				JMP START;			
			END_IF
		ELSE
			IF _Command.ExecuteDataReturn(ADR(_ExecutionParameters.CommandText), SIZEOF(_ExecutionParameters.CommandText), ADR(_SQLResult)) THEN
				IF _Command.bError THEN
					_GetError := TRUE;
					_Logger := _Command.ipTcResult;
					_State := DB_COMMAND_EXECUTION_STATE.DISCONNECTING;
				ELSE
					_State := DB_COMMAND_EXECUTION_STATE.LOADING_RESULT_DATA_SET;
				END_IF
				
				JMP START;			
			END_IF
		END_IF
		
	DB_COMMAND_EXECUTION_STATE.LOADING_RESULT_DATA_SET:
		IF _SQLResult.Read(0, _ExecutionParameters.MaxRecordsToReadAtTime, _ExecutionParameters.TargetBuffer, _ExecutionParameters.TargetBufferSize, TRUE, TRUE) THEN			
			IF _SQLResult.bError THEN
				_GetError := TRUE;
				_SQLResult.Release();
				_Logger := _SQLResult.ipTcResult;
			ELSE
				_DataSetLoaded := TRUE;
			END_IF

			_State := DB_COMMAND_EXECUTION_STATE.DISCONNECTING;
			
			JMP START;			
		END_IF

	DB_COMMAND_EXECUTION_STATE.DISCONNECTING:
		CASE _DisconnectingState OF
			DB_COMMAND_DISCONNECTING_STATE.IDLING:
				IF _DataSetLoaded THEN
					_DisconnectingState := DB_COMMAND_DISCONNECTING_STATE.DATA_SET_RELEASING;
				ELSIF _Connected THEN
					_DisconnectingState := DB_COMMAND_DISCONNECTING_STATE.DISCONNECTING;					
				ELSE
					_State := DB_COMMAND_EXECUTION_STATE.IDLING;	
					_Done := _LastException.Empty;	
				END_IF
				
				JMP START;
				
			DB_COMMAND_DISCONNECTING_STATE.DATA_SET_RELEASING:
				IF _SQLResult.Release() THEN
					_DataSetLoaded := FALSE;
					_DisconnectingState := DB_COMMAND_DISCONNECTING_STATE.DISCONNECTING;
					JMP START;										
				END_IF
				
			DB_COMMAND_DISCONNECTING_STATE.DISCONNECTING:
				IF _DbConnection.Disconnect() THEN
					_Connected := FALSE;
					_DisconnectingState := DB_COMMAND_DISCONNECTING_STATE.IDLING;
					JMP START;										
				END_IF
		END_CASE	
END_CASE
END_METHOD

{attribute 'monitoring' := 'call'}
{attribute 'OPC.UA.DA.Property' := '1'}
{attribute 'OPC.UA.DA.Access' := '1'}
PROPERTY LastException : REFERENCE TO Exception
GET
LastException REF= _LastException;
END_GET
END_PROPERTY

METHOD Reset
VAR_OUTPUT
	exception : Exception;
END_VAR
IF Busy THEN
	_LastExceptionHelper.Throw(0, "Previous command execution is not finished", __POUNAME(), ClassName, CurrentNamespace.Name, __POSITION()); 
	RETURN;
END_IF

_Done := FALSE;
_State := DB_COMMAND_EXECUTION_STATE.STARTING;
_GetError := FALSE;
_Logger := 0;	
_Connected := FALSE;
_DataSetLoaded := FALSE;
_DisconnectingState := DB_COMMAND_DISCONNECTING_STATE.IDLING;
_LastException.Clear();
END_METHOD

METHOD Start 
VAR_INPUT
	dbId : UDINT;
	commandText : Tc2_System.T_MaxString;
	targetBuffer : PVOID;
	targetBufferSize : UDINT;
	maxRecordsToReadAtTime : UINT;
END_VAR
VAR_OUTPUT
	exception : Exception;
END_VAR
VAR
	executionParameters : POINTER TO DB_COMMAND_EXECUTION_PARAMETERS;
END_VAR
IF Busy THEN
	_LastExceptionHelper.Throw(0, "Previous command execution is not finished", __POUNAME(), ClassName, CurrentNamespace.Name, __POSITION()); 
	RETURN;
END_IF

IF maxRecordsToReadAtTime > 0 AND_THEN (targetBuffer = 0 OR_ELSE targetBufferSize = 0) THEN
	_LastExceptionHelper.Throw(0, "Parameter 'maxRecordsToReadAtTime' is greater then zero, but 'targetBuffer' or 'targetBufferSize' has incorrect values", __POUNAME(), ClassName, CurrentNamespace.Name, __POSITION()); 
	RETURN;
END_IF

_ExecutionParameters.DbId := dbId;
_ExecutionParameters.CommandText := commandText;
_ExecutionParameters.TargetBuffer := targetBuffer; 
_ExecutionParameters.TargetBufferSize := targetBufferSize;
_ExecutionParameters.MaxRecordsToReadAtTime := maxRecordsToReadAtTime;

Reset();
END_METHOD

{attribute 'monitoring' := 'call'}
{attribute 'OPC.UA.DA.Property' := '1'}
{attribute 'OPC.UA.DA.Access' := '1'}
PROPERTY State : DB_COMMAND_EXECUTION_STATE
GET
State := _State;
END_GET
END_PROPERTY

{attribute 'monitoring' := 'call'}
{attribute 'OPC.UA.DA.Property' := '1'}
{attribute 'OPC.UA.DA.Access' := '1'}
PROPERTY Timeout : TIME
GET
Timeout := _Command.tTimeout;
END_GET
SET
_Command.tTimeout := Timeout;
_SQLResult.tTimeout := Timeout;
END_SET
END_PROPERTY

END_FUNCTION_BLOCK

// ---- Database/StoredProcedure/DbProcedureExecutor.TcPOU
{attribute 'no_explicit_call' := 'do not call this function block directly'} 
FUNCTION_BLOCK DbProcedureExecutor EXTENDS TC.ToolkitObject IMPLEMENTS TC.IAction
VAR	
	_ClassName : STRING := __POUNAME();

	_DbConnection : Tc3_Database.FB_SQLDatabaseEvt(sNetID := '', tTimeout := T#10S);	

	_ExecutionParameters : DB_ROCEDURE_EXECUTION_PARAMETERS;

	_StoredProcedure : Tc3_Database.FB_SQLStoredProcedureEvt(sNetID:='', tTimeout := T#10S);
	_SQLResult: Tc3_Database.FB_SQLResultEvt(sNetID := '', tTimeout := T#10S);
	
	_Done : BOOL;
	_State : DB_PROCEDURE_EXECUTION_STATE;
	_GetError : BOOL;
	_Logger : Tc3_EventLogger.I_TcMessage;	
	_Connected : BOOL;
	_Prepared : BOOL;
	_DataSetLoaded : BOOL;
	_DisconnectingState : DB_PROCEDURE_DISCONNECTING_STATE;
	_LastException : Exception;
END_VAR

{attribute 'monitoring' := 'call'}
{attribute 'OPC.UA.DA.Property' := '1'}
{attribute 'OPC.UA.DA.Access' := '1'}
PROPERTY Busy : BOOL
GET
Busy := State <> DB_PROCEDURE_EXECUTION_STATE.IDLING;
END_GET
END_PROPERTY

{attribute 'monitoring' := 'call'}
PROPERTY ClassName : STRING
GET
ClassName := _ClassName;
END_GET
END_PROPERTY

{attribute 'monitoring' := 'call'}
{attribute 'OPC.UA.DA.Property' := '1'}
{attribute 'OPC.UA.DA.Access' := '1'}
PROPERTY Done : BOOL
GET
Done := _Done;
END_GET
END_PROPERTY

{attribute 'monitoring' := 'call'}
{attribute 'OPC.UA.DA.Property' := '1'}
{attribute 'OPC.UA.DA.Access' := '1'}
PROPERTY Error : BOOL
GET
Error := State = DB_PROCEDURE_EXECUTION_STATE.IDLING AND_THEN NOT _LastException.Empty;
END_GET
END_PROPERTY

METHOD Execute
VAR
	requestEventTextError : BOOL;
	requestEventTextErrorCode : HRESULT;
END_VAR
VAR_INST
	errorMessage : STRING(255);	
END_VAR
START:

IF NOT _LastException.Empty THEN
	_GetError := FALSE;
END_IF

IF _GetError THEN
	IF _Logger <> 0 THEN 
		IF _Logger.RequestEventText(1033, errorMessage, SIZEOF(errorMessage), bError => requestEventTextError, hrErrorCode => requestEventTextErrorCode) THEN
			IF requestEventTextError THEN					
				errorMessage := StringHelper.Concat2('_Logger.RequestEventText() call error. Error code is ', TO_STRING(requestEventTextErrorCode));
			END_IF
		ELSE
			RETURN;
		END_IF			
	ELSE
		errorMessage :=  'Logger is not specified';
	END_IF				
	
	_LastExceptionHelper.Throw(0, TO_WSTRING(errorMessage), __POUNAME(), ClassName, CurrentNamespace.Name, __POSITION());
	JMP START;	
END_IF

CASE State OF
	DB_PROCEDURE_EXECUTION_STATE.STARTING:
		MEMSET(_ExecutionParameters.TargetBuffer, 0, _ExecutionParameters.TargetBufferSize);	
		_State := DB_PROCEDURE_EXECUTION_STATE.CONNECTING;			
		JMP START;
				
	DB_PROCEDURE_EXECUTION_STATE.CONNECTING:
		IF _DbConnection.Connect(hDBID := _ExecutionParameters.DBID) THEN
			IF _DbConnection.bError THEN
				_GetError := TRUE;
				_Logger := _DbConnection.ipTcResult;
				_State := DB_PROCEDURE_EXECUTION_STATE.DISCONNECTING;				
			ELSE
				_Connected := TRUE;
				_State := DB_PROCEDURE_EXECUTION_STATE.PREPARING;
			END_IF			

			JMP START;
		END_IF
	
	DB_PROCEDURE_EXECUTION_STATE.PREPARING:
		IF _DbConnection.CreateSP(sProcedureName := _ExecutionParameters.ProcedureName, pParameterInfo := _ExecutionParameters.ParameterDescriptors, cbParameterInfo := _ExecutionParameters.ParameterDescriptorsSize, pSQLProcedure := ADR(_StoredProcedure)) THEN
			IF _DbConnection.bError THEN
				_GetError := TRUE;
				_Logger := _DbConnection.ipTcResult;
				_State := DB_PROCEDURE_EXECUTION_STATE.DISCONNECTING;				
			ELSE
				_Prepared := TRUE;
				_State := DB_PROCEDURE_EXECUTION_STATE.EXECUTING;
			END_IF
			
			JMP START;
		END_IF
	
	DB_PROCEDURE_EXECUTION_STATE.EXECUTING:
		IF _ExecutionParameters.MaxRecordsToReadAtTime = 0 THEN
			IF _StoredProcedure.Execute(_ExecutionParameters.ParameterValues, _ExecutionParameters.ParameterValuesSize) THEN
				IF _StoredProcedure.bError THEN
					_GetError := TRUE;
					_Logger := _StoredProcedure.ipTcResult;
				END_IF
				
				_State := DB_PROCEDURE_EXECUTION_STATE.DISCONNECTING;
				
				JMP START;			
			END_IF
		ELSE
			IF _StoredProcedure.ExecuteDataReturn(_ExecutionParameters.ParameterValues, _ExecutionParameters.ParameterValuesSize, ADR(_SQLResult)) THEN
				IF _StoredProcedure.bError THEN
					_GetError := TRUE;
					_Logger := _StoredProcedure.ipTcResult;
					_State := DB_PROCEDURE_EXECUTION_STATE.DISCONNECTING;
				ELSE
					_State := DB_PROCEDURE_EXECUTION_STATE.LOADING_RESULT_DATA_SET;
				END_IF
								
				JMP START;			
			END_IF
		END_IF
		
	DB_PROCEDURE_EXECUTION_STATE.LOADING_RESULT_DATA_SET:
		IF _SQLResult.Read(0, _ExecutionParameters.MaxRecordsToReadAtTime, _ExecutionParameters.TargetBuffer, _ExecutionParameters.TargetBufferSize, TRUE, TRUE) THEN
			IF _SQLResult.bError THEN
				_GetError := TRUE;
				_SQLResult.Release();
				_Logger := _SQLResult.ipTcResult;
			ELSE				
				_DataSetLoaded := TRUE;
			END_IF
			
			_State := DB_PROCEDURE_EXECUTION_STATE.DISCONNECTING;
			
			JMP START;			
		END_IF		

	DB_PROCEDURE_EXECUTION_STATE.DISCONNECTING:
		CASE _DisconnectingState OF
			DB_PROCEDURE_DISCONNECTING_STATE.IDLING:				
				IF _DataSetLoaded THEN
					_DisconnectingState := DB_PROCEDURE_DISCONNECTING_STATE.DATA_SET_RELEASING;
				ELSIF _Prepared THEN
					_DisconnectingState := DB_PROCEDURE_DISCONNECTING_STATE.PARAMETERS_RELEASING;					
				ELSIF _Connected THEN
					_DisconnectingState := DB_PROCEDURE_DISCONNECTING_STATE.DISCONNECTING;					
				ELSE
					_State := DB_PROCEDURE_EXECUTION_STATE.IDLING;				
					_Done := _LastException.Empty;	
				END_IF
				
				JMP START;
				
			DB_PROCEDURE_DISCONNECTING_STATE.DATA_SET_RELEASING:
				IF _SQLResult.Release() THEN
					_DataSetLoaded := FALSE;
					_DisconnectingState := DB_PROCEDURE_DISCONNECTING_STATE.PARAMETERS_RELEASING;
					JMP START;					
				END_IF
			
			DB_PROCEDURE_DISCONNECTING_STATE.PARAMETERS_RELEASING:
				IF _StoredProcedure.Release() THEN
					_Prepared := FALSE;
					_DisconnectingState := DB_PROCEDURE_DISCONNECTING_STATE.DISCONNECTING;
					JMP START;										
				END_IF
				
			DB_PROCEDURE_DISCONNECTING_STATE.DISCONNECTING:
				IF _DbConnection.Disconnect() THEN
					_Connected := FALSE;
					_DisconnectingState := DB_PROCEDURE_DISCONNECTING_STATE.IDLING;
					JMP START;										
				END_IF
		END_CASE	
END_CASE
END_METHOD

{attribute 'monitoring' := 'call'}
{attribute 'OPC.UA.DA.Property' := '1'}
{attribute 'OPC.UA.DA.Access' := '1'}
PROPERTY LastException : REFERENCE TO Exception
GET
LastException REF= _LastException;
END_GET
END_PROPERTY

{attribute 'OPC.UA.DA.Property' := '1'}
{attribute 'OPC.UA.DA.Access' := '1'}
{attribute 'monitoring' := 'call'}
PROPERTY ProcedureName : REFERENCE TO Tc2_System.T_MaxString
GET
ProcedureName REF= _ExecutionParameters.ProcedureName;
END_GET
END_PROPERTY

METHOD Reset 
VAR_OUTPUT
	exception : Exception;
END_VAR
IF Busy THEN
	_LastExceptionHelper.Throw(0, "Previous command execution is not finished", __POUNAME(), ClassName, CurrentNamespace.Name, __POSITION()); 
	RETURN;
END_IF

_Done := FALSE;
_State := DB_PROCEDURE_EXECUTION_STATE.STARTING;
_GetError := FALSE;
_Logger := 0;	
_Connected := FALSE;
_Prepared := FALSE;
_DataSetLoaded := FALSE;
_DisconnectingState := DB_PROCEDURE_DISCONNECTING_STATE.IDLING;
_LastException.Clear();
END_METHOD

METHOD Start 
VAR_INPUT
	dbId : UDINT;
	procedureName : Tc2_System.T_MaxString;
	parameterDescriptors : POINTER TO Tc3_Database.ST_SQLSPParameter;
	parameterDescriptorsSize : UDINT;
	parameterValues : PVOID;
	parameterValuesSize : UDINT;
	targetBuffer : PVOID;
	targetBufferSize : UDINT;
	maxRecordsToReadAtTime : UINT;
END_VAR
VAR_OUTPUT
	exception : Exception;
END_VAR
IF Busy THEN
	_LastExceptionHelper.Throw(0, "Previous command execution is not finished", __POUNAME(), ClassName, CurrentNamespace.Name, __POSITION()); 
	RETURN;
END_IF

IF maxRecordsToReadAtTime > 0 AND_THEN (targetBuffer = 0 OR_ELSE targetBufferSize = 0) THEN
	_LastExceptionHelper.Throw(0, "Parameter 'maxRecordsToReadAtTime' is greater then zero, but 'targetBuffer' or 'targetBufferSize' has incorrect values", __POUNAME(), ClassName, CurrentNamespace.Name, __POSITION()); 
	RETURN;
END_IF

_ExecutionParameters.DbId := dbId;
_ExecutionParameters.ProcedureName := procedureName;
_ExecutionParameters.ParameterDescriptors := parameterDescriptors;
_ExecutionParameters.ParameterDescriptorsSize := parameterDescriptorsSize;
_ExecutionParameters.ParameterValues := parameterValues;
_ExecutionParameters.ParameterValuesSize := parameterValuesSize;
_ExecutionParameters.TargetBuffer := targetBuffer; 
_ExecutionParameters.TargetBufferSize := targetBufferSize;
_ExecutionParameters.MaxRecordsToReadAtTime := maxRecordsToReadAtTime;

Reset();
END_METHOD

{attribute 'monitoring' := 'call'}
{attribute 'OPC.UA.DA.Property' := '1'}
{attribute 'OPC.UA.DA.Access' := '1'}
PROPERTY State : DB_PROCEDURE_EXECUTION_STATE
GET
State := _State;
END_GET
END_PROPERTY

{attribute 'monitoring' := 'call'}
{attribute 'OPC.UA.DA.Property' := '1'}
{attribute 'OPC.UA.DA.Access' := '1'}
PROPERTY Timeout : TIME
GET
Timeout := _StoredProcedure.tTimeout;
END_GET
SET
_StoredProcedure.tTimeout := Timeout;
_SQLResult.tTimeout := Timeout;
END_SET
END_PROPERTY

END_FUNCTION_BLOCK

// ---- Files/CreateDirectory.TcPOU
{attribute 'no_explicit_call' := 'do not call this function block directly'} 
FUNCTION_BLOCK CreateDirectory EXTENDS ToolkitObject IMPLEMENTS IAction
VAR
	{attribute 'OPC.UA.DA' := '0'}
	_ClassName : STRING := __POUNAME();

	{attribute 'OPC.UA.DA' := '0'}
    _CreateDirectory : Tc2_System.FB_CreateDir;
	
	{attribute 'OPC.UA.DA' := '0'}
	_NeedStart : BOOL;
	{attribute 'OPC.UA.DA' := '0'}
	_Done : BOOL;
END_VAR

{attribute 'monitoring' := 'call'}
{attribute 'OPC.UA.DA.Property' := '1'}
{attribute 'OPC.UA.DA' := '1'}
PROPERTY AmsNetId : Tc2_System.T_AmsNetID
GET
AmsNetId := _CreateDirectory.sNetId;
END_GET
SET
_CreateDirectory.sNetId := AmsNetId;
END_SET
END_PROPERTY

{attribute 'monitoring' := 'call'}
{attribute 'OPC.UA.DA.Property' := '1'}
{attribute 'OPC.UA.DA.Access' := '1'}
PROPERTY Busy : BOOL
GET
Busy := _NeedStart OR_ELSE _CreateDirectory.bBusy;
END_GET
END_PROPERTY

{attribute 'monitoring' := 'call'}
PROPERTY ClassName : STRING
GET
ClassName := _ClassName;
END_GET
END_PROPERTY

{attribute 'monitoring' := 'call'}
{attribute 'OPC.UA.DA.Property' := '1'}
{attribute 'OPC.UA.DA.Access' := '1'}
PROPERTY Done : BOOL
GET
Done := _Done;
END_GET
END_PROPERTY

{attribute 'monitoring' := 'call'}
{attribute 'OPC.UA.DA.Property' := '1'}
{attribute 'OPC.UA.DA.Access' := '1'}
PROPERTY Error : BOOL
GET
Error := _CreateDirectory.bError;
END_GET
END_PROPERTY

METHOD Execute
VAR
	message : ERROR_MESSAGE;
END_VAR
IF _NeedStart OR_ELSE _CreateDirectory.bBusy THEN
	_CreateDirectory(bExecute := TRUE);
	_NeedStart := FALSE;
	
	IF _CreateDirectory.bError THEN
		message := "An error occurred while creating the directory '";
		WStringHelper.Append2(message, TO_WSTRING(_CreateDirectory.sPathName), "'");	
		_LastException.Configure(message, __POUNAME(), ClassName, CurrentNamespace.Name, __POSITION(), _CreateDirectory.nErrId).Throw();
	ELSIF NOT _CreateDirectory.bBusy THEN
		_Done := TRUE;
	END_IF
END_IF
END_METHOD

{attribute 'monitoring' := 'call'}
{attribute 'OPC.UA.DA.Property' := '1'}
{attribute 'OPC.UA.DA.Access' := '1'}
PROPERTY LastException : REFERENCE TO Exception
GET
LastException REF= _LastException;
END_GET
END_PROPERTY

{attribute 'monitoring' := 'call'}
{attribute 'OPC.UA.DA.Property' := '1'}
{attribute 'OPC.UA.DA' := '1'}
PROPERTY PathType : Tc2_System.E_OpenPath
GET
PathType := _CreateDirectory.ePath;
END_GET
SET
_CreateDirectory.ePath := PathType;
END_SET
END_PROPERTY

METHOD Start
VAR_INPUT
	directoryPath : Tc2_System.T_MaxString;
END_VAR
_NeedStart := TRUE;
_Done := FALSE;
_CreateDirectory.sPathName := directoryPath;

_LastException.Clear();
END_METHOD

{attribute 'monitoring' := 'call'}
{attribute 'OPC.UA.DA.Property' := '1'}
{attribute 'OPC.UA.DA' := '1'}
PROPERTY Timeout : TIME
GET
Timeout := _CreateDirectory.tTimeout;
END_GET
SET
_CreateDirectory.tTimeout := Timeout;
END_SET
END_PROPERTY

END_FUNCTION_BLOCK

// ---- Files/DeleteDirectory.TcPOU
{attribute 'no_explicit_call' := 'do not call this function block directly'} 
FUNCTION_BLOCK DeleteDirectory EXTENDS ToolkitObject IMPLEMENTS IAction
VAR
	{attribute 'OPC.UA.DA' := '0'}
	_ClassName : STRING := __POUNAME();

	{attribute 'OPC.UA.DA' := '0'}
    _DeleteDirectory : Tc2_System.FB_RemoveDir;	
	
	{attribute 'OPC.UA.DA' := '0'}
	_NeedStart : BOOL;
	{attribute 'OPC.UA.DA' := '0'}
	_Done : BOOL;
END_VAR

{attribute 'monitoring' := 'call'}
{attribute 'OPC.UA.DA.Property' := '1'}
{attribute 'OPC.UA.DA' := '1'}
PROPERTY AmsNetId : Tc2_System.T_AmsNetID
GET
AmsNetId := _DeleteDirectory.sNetId;
END_GET
SET
_DeleteDirectory.sNetId := AmsNetId;
END_SET
END_PROPERTY

{attribute 'monitoring' := 'call'}
{attribute 'OPC.UA.DA.Property' := '1'}
{attribute 'OPC.UA.DA.Access' := '1'}
PROPERTY Busy : BOOL
GET
Busy := _NeedStart OR_ELSE _DeleteDirectory.bBusy;
END_GET
END_PROPERTY

{attribute 'monitoring' := 'call'}
PROPERTY ClassName : STRING
GET
ClassName := _ClassName;
END_GET
END_PROPERTY

{attribute 'monitoring' := 'call'}
{attribute 'OPC.UA.DA.Property' := '1'}
{attribute 'OPC.UA.DA.Access' := '1'}
PROPERTY Done : BOOL
GET
Done := _Done;
END_GET
END_PROPERTY

{attribute 'monitoring' := 'call'}
{attribute 'OPC.UA.DA.Property' := '1'}
{attribute 'OPC.UA.DA.Access' := '1'}
PROPERTY Error : BOOL
GET
Error := _DeleteDirectory.bError;
END_GET
END_PROPERTY

METHOD Execute
VAR
	errorMessage : ERROR_MESSAGE;
END_VAR
IF _NeedStart OR_ELSE _DeleteDirectory.bBusy THEN
	_DeleteDirectory(bExecute := TRUE);
	_NeedStart := FALSE;
	
	IF _DeleteDirectory.bError THEN
		errorMessage := "An error occurred while deleting the directory '";
		WStringHelper.Append2(errorMessage, TO_WSTRING(_DeleteDirectory.sPathName), "'");	
		_LastException.Configure(errorMessage, __POUNAME(), ClassName, CurrentNamespace.Name, __POSITION(), _DeleteDirectory.nErrId).Throw();
	ELSIF NOT _DeleteDirectory.bBusy THEN
		_Done := TRUE;
	END_IF
END_IF
END_METHOD

{attribute 'monitoring' := 'call'}
{attribute 'OPC.UA.DA.Property' := '1'}
{attribute 'OPC.UA.DA.Access' := '1'}
PROPERTY LastException : REFERENCE TO Exception
GET
LastException REF= _LastException;
END_GET
END_PROPERTY

{attribute 'monitoring' := 'call'}
{attribute 'OPC.UA.DA.Property' := '1'}
{attribute 'OPC.UA.DA' := '1'}
PROPERTY PathType : Tc2_System.E_OpenPath
GET
PathType := _DeleteDirectory.ePath;
END_GET
SET
_DeleteDirectory.ePath := PathType;
END_SET
END_PROPERTY

METHOD Start
VAR_INPUT
	directoryPath : Tc2_System.T_MaxString;
END_VAR
_NeedStart := TRUE;
_Done := FALSE;
_DeleteDirectory.sPathName := directoryPath;

_LastException.Clear();
END_METHOD

{attribute 'monitoring' := 'call'}
{attribute 'OPC.UA.DA.Property' := '1'}
{attribute 'OPC.UA.DA' := '1'}
PROPERTY Timeout : TIME
GET
Timeout := _DeleteDirectory.tTimeout;
END_GET
SET
_DeleteDirectory.tTimeout := Timeout;
END_SET
END_PROPERTY

END_FUNCTION_BLOCK

// ---- Files/DeleteFile.TcPOU
{attribute 'no_explicit_call' := 'do not call this function block directly'} 
FUNCTION_BLOCK DeleteFile EXTENDS ToolkitObject IMPLEMENTS IAction
VAR
	{attribute 'OPC.UA.DA' := '0'}
	_ClassName : STRING := __POUNAME();

	{attribute 'OPC.UA.DA' := '0'}
    _Delete : Tc2_System.FB_FileDelete;
	
	{attribute 'OPC.UA.DA' := '0'}
	_NeedStart : BOOL;
	{attribute 'OPC.UA.DA' := '0'}
	_Done : BOOL;
END_VAR

{attribute 'monitoring' := 'call'}
{attribute 'OPC.UA.DA.Property' := '1'}
{attribute 'OPC.UA.DA' := '1'}
PROPERTY AmsNetId : Tc2_System.T_AmsNetID
GET
AmsNetId := _Delete.sNetId;
END_GET
SET
_Delete.sNetId := AmsNetId;
END_SET
END_PROPERTY

{attribute 'monitoring' := 'call'}
{attribute 'OPC.UA.DA.Property' := '1'}
{attribute 'OPC.UA.DA.Access' := '1'}
PROPERTY Busy : BOOL
GET
Busy := _NeedStart OR_ELSE _Delete.bBusy;
END_GET
END_PROPERTY

{attribute 'monitoring' := 'call'}
PROPERTY ClassName : STRING
GET
ClassName := _ClassName;
END_GET
END_PROPERTY

{attribute 'monitoring' := 'call'}
{attribute 'OPC.UA.DA.Property' := '1'}
{attribute 'OPC.UA.DA.Access' := '1'}
PROPERTY Done : BOOL
GET
Done := _Done;
END_GET
END_PROPERTY

{attribute 'monitoring' := 'call'}
{attribute 'OPC.UA.DA.Property' := '1'}
{attribute 'OPC.UA.DA.Access' := '1'}
PROPERTY Error : BOOL
GET
Error := _Delete.bError;
END_GET
END_PROPERTY

METHOD Execute
VAR
	message : ERROR_MESSAGE;
END_VAR
IF _NeedStart OR_ELSE _Delete.bBusy THEN
	_Delete(bExecute := TRUE);
	_NeedStart := FALSE;
	
	IF _Delete.bError THEN
		message := "An error occurred while creating the file '";
		WStringHelper.Append2(message, TO_WSTRING(_Delete.sPathName), "'");	
		_LastException.Configure(message, __POUNAME(), ClassName, CurrentNamespace.Name, __POSITION(), _Delete.nErrId).Throw();
	ELSIF NOT _Delete.bBusy THEN
		_Done := TRUE;
	END_IF
END_IF
END_METHOD

{attribute 'monitoring' := 'call'}
{attribute 'OPC.UA.DA.Property' := '1'}
{attribute 'OPC.UA.DA.Access' := '1'}
PROPERTY LastException : REFERENCE TO Exception
GET
LastException REF= _LastException;
END_GET
END_PROPERTY

{attribute 'monitoring' := 'call'}
{attribute 'OPC.UA.DA.Property' := '1'}
{attribute 'OPC.UA.DA' := '1'}
PROPERTY PathType : Tc2_System.E_OpenPath
GET
PathType := _Delete.ePath;
END_GET
SET
_Delete.ePath := PathType;
END_SET
END_PROPERTY

METHOD Start
VAR_INPUT
	filePath : Tc2_System.T_MaxString;
END_VAR
_NeedStart := TRUE;
_Done := FALSE;
_Delete.sPathName := filePath;

_LastException.Clear();
END_METHOD

{attribute 'monitoring' := 'call'}
{attribute 'OPC.UA.DA.Property' := '1'}
{attribute 'OPC.UA.DA' := '1'}
PROPERTY Timeout : TIME
GET
Timeout := _Delete.tTimeout;
END_GET
SET
_Delete.tTimeout := Timeout;
END_SET
END_PROPERTY

END_FUNCTION_BLOCK

// ---- Files/FileContentManager/FileContentManager.TcPOU
{attribute 'no_explicit_call' := 'do not call this function block directly'} 
FUNCTION_BLOCK FileContentManager EXTENDS ToolkitObject IMPLEMENTS IAbortableProcess
VAR
	_ClassName : STRING := __POUNAME();

	_FilePath : Tc2_System.T_MaxString;	
	_OpenMode : FILE_OPEN_MODE;
	_ContentHandlingMode : FILE_CONTENT_HANDLING_MODE;
	_PathType : E_OpenPath;	
	_AmsNetId : Tc2_System.T_AmsNetID;
	_FileHandle : UINT;
		
	_TaskExecutor : SequentialTaskExecutor;
END_VAR

{attribute 'monitoring' := 'call'}
{attribute 'OPC.UA.DA.Property' := '1'}
{attribute 'OPC.UA.DA.Access' := '1'}
PROPERTY FINAL Aborted : BOOL
GET
Aborted := _TaskExecutor.Aborted;
END_GET
END_PROPERTY

{attribute 'monitoring' := 'call'}
{attribute 'OPC.UA.DA.Property' := '1'}
{attribute 'OPC.UA.DA.Access' := '1'}
PROPERTY FINAL Aborting : BOOL
GET
Busy := _TaskExecutor.Busy;
END_GET
END_PROPERTY

{attribute 'monitoring' := 'call'}
{attribute 'OPC.UA.DA.Property' := '1'}
{attribute 'OPC.UA.DA.Access' := '1'}
PROPERTY AbortReason : REFERENCE TO ERROR_MESSAGE
GET
AbortReason REF= _TaskExecutor.AbortReason;
END_GET
END_PROPERTY

METHOD AddTask
VAR_INPUT
	fileOperation : REFERENCE TO FileContentTask;
END_VAR
IF __ISVALIDREF(fileOperation) THEN
	fileOperation.FileContentManager REF= THIS^;

	_TaskExecutor.AddTask(fileOperation);
END_IF
END_METHOD

{attribute 'monitoring' := 'call'}
{attribute 'OPC.UA.DA.Property' := '1'}
PROPERTY AmsNetId : Tc2_System.T_AmsNetID
GET
AmsNetId := _AmsNetId;
END_GET
SET
_AmsNetId := AmsNetId;
END_SET
END_PROPERTY

{attribute 'monitoring' := 'call'}
{attribute 'OPC.UA.DA.Property' := '1'}
{attribute 'OPC.UA.DA.Access' := '1'}
PROPERTY FINAL Busy : BOOL
GET
Busy := _TaskExecutor.Busy;
END_GET
END_PROPERTY

{attribute 'monitoring' := 'call'}
PROPERTY ClassName : STRING
GET
ClassName := _ClassName;
END_GET
END_PROPERTY

{attribute 'monitoring' := 'call'}
{attribute 'OPC.UA.DA.Property' := '1'}
{attribute 'OPC.UA.DA.Access' := '1'}
PROPERTY ContentHandlingMode : FILE_CONTENT_HANDLING_MODE
GET
ContentHandlingMode := _ContentHandlingMode;
END_GET
SET // INTERNAL
_ContentHandlingMode := ContentHandlingMode;
END_SET
END_PROPERTY

{attribute 'monitoring' := 'call'}
{attribute 'OPC.UA.DA.Property' := '1'}
{attribute 'OPC.UA.DA.Access' := '1'}
PROPERTY FINAL Error : BOOL
GET
Error := _TaskExecutor.Error;
END_GET
END_PROPERTY

{attribute 'monitoring' := 'call'}
{attribute 'OPC.UA.DA.Property' := '1'}
{attribute 'OPC.UA.DA.Access' := '1'}
PROPERTY FINAL ErrorMessage : REFERENCE TO Exception
GET
ErrorMessage REF= _TaskExecutor.ErrorMessage;
END_GET
END_PROPERTY

METHOD Execute
_TaskExecutor.Execute();
END_METHOD

METHOD FB_exit : BOOL
VAR_INPUT
	bInCopyCode : BOOL; // if TRUE, the exit method is called for exiting an instance that is copied afterwards (online change).
END_VAR
VAR_INST
	_Close : Tc2_System.FB_FileClose;
END_VAR
IF _FileHandle <> 0 THEN
	_Close(
		bExecute := TRUE,
		hFile := _FileHandle,
		sNetId := _AmsNetId,
		tTimeout := T#1S		
	); 
END_IF
END_METHOD

METHOD FB_init : BOOL
VAR_INPUT
	bInitRetains : BOOL; // if TRUE, the retain variables are initialized (warm start / cold start)
	bInCopyCode : BOOL; // if TRUE, the instance afterwards gets moved into the copy code (online change)
END_VAR
_TaskExecutor.ContinueOnTaskError := TRUE;
END_METHOD

PROPERTY FileHandle : UINT
GET
FileHandle := _FileHandle;
END_GET
SET // INTERNAL
_FileHandle := FileHandle;
END_SET
END_PROPERTY

{attribute 'monitoring' := 'call'}
{attribute 'OPC.UA.DA.Property' := '1'}
{attribute 'OPC.UA.DA.Access' := '1'}
PROPERTY FilePath : Tc2_System.T_MaxString
GET
FilePath := _FilePath;
END_GET
SET // INTERNAL
_FilePath := FilePath;
END_SET
END_PROPERTY

{attribute 'monitoring' := 'call'}
{attribute 'OPC.UA.DA.Property' := '1'}
{attribute 'OPC.UA.DA.Access' := '1'}
PROPERTY IsOpen : BOOL
GET
IsOpen := _FileHandle <> 0;
END_GET
END_PROPERTY

{attribute 'monitoring' := 'call'}
{attribute 'OPC.UA.DA.Property' := '1'}
{attribute 'OPC.UA.DA.Access' := '1'}
PROPERTY OpenMode : FILE_OPEN_MODE
GET
OpenMode := _OpenMode;
END_GET
SET // INTERNAL
_OpenMode := OpenMode;
END_SET
END_PROPERTY

{attribute 'monitoring' := 'call'}
{attribute 'OPC.UA.DA.Property' := '1'}
{attribute 'OPC.UA.DA.Access' := '1'}
PROPERTY PathType : E_OpenPath
GET
PathType := _PathType;
END_GET
SET // INTERNAL
_PathType := PathType;
END_SET
END_PROPERTY

METHOD RequestAbort
VAR_INPUT 
	reason : ERROR_MESSAGE;
END_VAR
_TaskExecutor.RequestAbort(reason);
END_METHOD

METHOD Start
_TaskExecutor.Start();
END_METHOD

END_FUNCTION_BLOCK

// ---- Tasks/SequentialTaskExecutor.TcPOU
{attribute 'no_explicit_call' := 'do not call this function block directly'} 
FUNCTION_BLOCK SequentialTaskExecutor EXTENDS ToolkitObject IMPLEMENTS IAbortableProcess
VAR
	_ClassName : STRING := __POUNAME();

	_Tasks : List(POINTER_TYPE.OBJECT_POINTER); // of POINTER TO Task  
	
	_ContinueOnTaskError : BOOL;

	_Busy : BOOL;
	_AbortRequested : BOOL;
	_Aborted : BOOL;
	_Error : BOOL;
	_ErrorMessage : ERROR_MESSAGE;
	_AbortReason : ERROR_MESSAGE;
END_VAR

{attribute 'monitoring' := 'call'}
{attribute 'OPC.UA.DA.Property' := '1'}
{attribute 'OPC.UA.DA.Access' := '1'}
PROPERTY FINAL Aborted : BOOL
GET
Aborted := _Aborted;
END_GET
END_PROPERTY

{attribute 'monitoring' := 'call'}
{attribute 'OPC.UA.DA.Property' := '1'}
{attribute 'OPC.UA.DA.Access' := '1'}
PROPERTY AbortReason : REFERENCE TO ERROR_MESSAGE
GET
AbortReason REF= _AbortReason;
END_GET
END_PROPERTY

METHOD AddTask
VAR_INPUT
	task : REFERENCE TO Task; // instance should be managed by external logic
END_VAR
IF NOT __ISVALIDREF(task) THEN
	RETURN;
END_IF

_Tasks.Append(ADR(task));
END_METHOD

{attribute 'monitoring' := 'call'}
{attribute 'OPC.UA.DA.Property' := '1'}
{attribute 'OPC.UA.DA.Access' := '1'}
PROPERTY FINAL Busy : BOOL
GET
Busy := _Busy;
END_GET
END_PROPERTY

{attribute 'monitoring' := 'call'}
PROPERTY ClassName : STRING
GET
ClassName := _ClassName;
END_GET
END_PROPERTY

METHOD ClearInactiveTasks
VAR
	i : DINT;
	task : POINTER TO Task;
END_VAR
FOR i := _Tasks.Count - 1 TO 0 BY -1 DO
	IF i = 0 THEN
		task := _Tasks.Get(0);
		
		IF task^.State = TASK_STATE.EXECUTING OR_ELSE task^.State = TASK_STATE.ABORTING THEN
			CONTINUE;			
		END_IF
	END_IF
	
	_Tasks.RemoveAt(i, FALSE);
END_FOR
END_METHOD

{attribute 'monitoring' := 'call'}
{attribute 'OPC.UA.DA.Property' := '1'}
{attribute 'OPC.UA.DA.Access' := '1'}
PROPERTY FINAL ContinueOnTaskError : BOOL
GET
ContinueOnTaskError := _ContinueOnTaskError;
END_GET
SET
_ContinueOnTaskError := ContinueOnTaskError;
END_SET
END_PROPERTY

{attribute 'monitoring' := 'call'}
{attribute 'OPC.UA.DA.Property' := '1'}
{attribute 'OPC.UA.DA.Access' := '1'}
PROPERTY FINAL Error : BOOL
GET
Error := _Error;
END_GET
END_PROPERTY

{attribute 'monitoring' := 'call'}
{attribute 'OPC.UA.DA.Property' := '1'}
{attribute 'OPC.UA.DA.Access' := '1'}
PROPERTY FINAL ErrorMessage : REFERENCE TO ERROR_MESSAGE
GET
ErrorMessage REF= _ErrorMessage;
END_GET
END_PROPERTY

METHOD Execute 
VAR
	task : POINTER TO Task;
	taskManagerAbortMessage : ERROR_MESSAGE := "TaskManager aborted with reason: ";
END_VAR
START:

IF NOT Busy OR_ELSE _Tasks.Count = 0 THEN
	RETURN;
END_IF

task := _Tasks.Get(0);

__TRY
	CASE task^.State OF
		TASK_STATE.EXECUTING:
			IF _AbortRequested THEN
				_AbortRequested := FALSE;
				
				IF task^.RequestAbort(TRUE) THEN
					task^.State := TASK_STATE.ABORTED;
				ELSE
					RETURN;
				END_IF
			ELSE
				IF task^.Execute(FALSE) THEN
					task^.State := TASK_STATE.DONE;
				ELSE
					RETURN;
				END_IF		
			END_IF

			_Tasks.Remove(task, FALSE);
							
		TASK_STATE.ABORTING:
			IF task^.RequestAbort(FALSE) THEN
				task^.State := TASK_STATE.ABORTED;
				
				_Tasks.Remove(task, FALSE);
			ELSE
				RETURN;
			END_IF
		ELSE
			task^.AbortReason := "";
			task^.ErrorMessage := "";
			
			IF task^.Execute(TRUE) THEN
				task^.State := TASK_STATE.DONE;

				_Tasks.Remove(task, FALSE);
			ELSE
				RETURN;
			END_IF
	END_CASE	
	
	_Tasks.Remove(task, FALSE);	
__CATCH
	task^.ErrorMessage := ExceptionHelper.LastException.ToString(FALSE);
	task^.State := TASK_STATE.ERROR;
	
	_Tasks.Remove(task, FALSE);

	IF NOT ContinueOnTaskError THEN
		setError(ExceptionHelper.LastException.ToString(FALSE));		
		ExceptionHelper.LastException.Throw();
	END_IF	
__ENDTRY

JMP START;
END_METHOD

METHOD RequestAbort
VAR_INPUT 
	reason : ERROR_MESSAGE;
END_VAR
VAR
	task : POINTER TO Task;
END_VAR
IF Busy THEN	
	_AbortReason := reason;
	
	IF _Tasks.Count > 0 THEN
		task := _Tasks.Get(0);
		
		IF task^.State = TASK_STATE.EXECUTING THEN
			_AbortRequested := TRUE;
			RETURN;
		END_IF
	END_IF

	setAborted();
END_IF
END_METHOD

METHOD PRIVATE setAborted
_Busy := FALSE;
_AbortRequested := FALSE;
_Aborted := TRUE;
_Error := FALSE;
END_METHOD

METHOD PRIVATE setBusy
_Busy := TRUE;
_AbortRequested := FALSE;
_Aborted := FALSE;
_Error := FALSE;
END_METHOD

METHOD PRIVATE setError
VAR_IN_OUT CONSTANT
	errorMessage : ERROR_MESSAGE;
END_VAR
_Busy := FALSE;
_AbortRequested := FALSE;
_Aborted := FALSE;
_Error := TRUE;

IF __ISVALIDREF(errorMessage) THEN
	_ErrorMessage := errorMessage;
END_IF
END_METHOD

METHOD Start
IF Busy THEN
	//exceptionFactory.ThrowException(__POSITION(), "Task manager in aborting state", __POUNAME(), ClassName, CurrentNamespace.Name, __POSITION()).Throw();
END_IF

_ErrorMessage := "";
_AbortReason := "";
setBusy();

Start := TRUE;
END_METHOD

END_FUNCTION_BLOCK

// ---- Tasks/Task.TcPOU
{attribute 'no_explicit_call' := 'do not call this function block directly'} 
FUNCTION_BLOCK ABSTRACT Task EXTENDS ToolkitObject
VAR
	_State : TASK_STATE;
	_ErrorMessage : ERROR_MESSAGE;
	_AbortReason : ERROR_MESSAGE;
END_VAR

{attribute 'monitoring' := 'call'}
{attribute 'OPC.UA.DA.Property' := '1'}
{attribute 'OPC.UA.DA.Access' := '1'}
PROPERTY FINAL AbortReason : REFERENCE TO ERROR_MESSAGE
GET
Abortreason REF= _AbortReason;
END_GET
END_PROPERTY

{attribute 'monitoring' := 'call'}
{attribute 'OPC.UA.DA.Property' := '1'}
{attribute 'OPC.UA.DA.Access' := '1'}
PROPERTY FINAL ErrorMessage : REFERENCE TO ERROR_MESSAGE
GET
ErrorMessage REF= _ErrorMessage;
END_GET
END_PROPERTY

METHOD Execute : BOOL
VAR_INPUT
	start : BOOL;
END_VAR
END_METHOD

METHOD OnStateChanged
VAR_INPUT
	oldState : TASK_STATE;
END_VAR
END_METHOD

METHOD OnStateChanging
VAR_INPUT
	newState : TASK_STATE;
END_VAR
END_METHOD

METHOD ABSTRACT RequestAbort : BOOL
VAR_INPUT
	start : BOOL;
END_VAR
END_METHOD

{attribute 'monitoring' := 'call'}
{attribute 'OPC.UA.DA.Property' := '1'}
{attribute 'OPC.UA.DA.Access' := '1'}
PROPERTY FINAL State : TASK_STATE
GET
State := _State;
END_GET
SET // INTERNAL
VAR
	oldState : TASK_STATE;
END_VAR
IF _State <> State THEN
	oldState := _State;
	
	OnStateChanging(State);
	_State := State;
	OnStateChanged(oldState);
END_IF
END_SET
END_PROPERTY

END_FUNCTION_BLOCK

// ---- Files/FileContentManager/FileContentTask.TcPOU
{attribute 'enable_dynamic_creation'}	
{attribute 'no_explicit_call' := 'do not call this function block directly'} 
FUNCTION_BLOCK ABSTRACT FileContentTask EXTENDS Task
VAR_INPUT
 	Timeout : TIME := T#2S;
END_VAR
VAR
	_FileContentManager : REFERENCE TO FileContentManager; 
END_VAR

PROPERTY INTERNAL FileContentManager : REFERENCE TO FileContentManager
GET
FileContentManager REF= _FileContentManager;
END_GET
SET
_FileContentManager REF= FileContentManager;
END_SET
END_PROPERTY

METHOD PROTECTED GetErrorMessageByErrorId : WSTRING(255)
VAR_INPUT
	errorId : UDINT;
END_VAR
CASE errorId OF
	1795: GetErrorMessageByErrorId := "invalid or unknown file handle";
	1802: GetErrorMessageByErrorId := "no memory for read buffer";
	1804: GetErrorMessageByErrorId := "file not found";
	1806: GetErrorMessageByErrorId := "file was opened with wrong method";
	1827: GetErrorMessageByErrorId := "folder already exists or invalid sPathName or ePath parameter";
END_CASE

IF GetErrorMessageByErrorId <> "" THEN
	GetErrorMessageByErrorId := WStringHelper.Concat2(": ", GetErrorMessageByErrorId);
END_IF
END_METHOD

METHOD RequestAbort : BOOL
VAR_INPUT
	start : BOOL;
END_VAR
IF Execute(start) = EXECUTION_STATE.BUSY THEN
	RequestAbort := EXECUTION_STATE.BUSY;
ELSE
	RequestAbort := EXECUTION_STATE.DONE;
END_IF
END_METHOD

METHOD PROTECTED Validate
VAR
	//exceptionFactory : ExceptionFactory(__POUNAME(), ClassName, CurrentNamespace.Name);
END_VAR
IF NOT __ISVALIDREF(FileContentManager) THEN
	//exceptionFactory.ThrowException(__POSITION(), "File content menager is not specified");
END_IF

IF FileContentManager.FileHandle = 0 THEN
	//exceptionFactory.ThrowException(__POSITION(), "File is not open");
END_IF
END_METHOD

END_FUNCTION_BLOCK

// ---- Files/FileContentManager/Tasks/FileCloseTask.TcPOU
{attribute 'enable_dynamic_creation'}	
{attribute 'no_explicit_call' := 'do not call this function block directly'} 
FUNCTION_BLOCK FileCloseTask EXTENDS FileContentTask
VAR
	_ClassName : STRING := __POUNAME();

    _Close : Tc2_System.FB_FileClose;
END_VAR

{attribute 'monitoring' := 'call'}
PROPERTY ClassName : STRING
GET
ClassName := _ClassName;
END_GET
END_PROPERTY

METHOD Execute : BOOL
VAR_INPUT
	start : BOOL;
END_VAR
VAR
	//exceptionFactory : ExceptionFactory(__POUNAME(), ClassName, CurrentNamespace.Name);
END_VAR
IF start THEN
	Validate();

	_Close(
		bExecute := FALSE,
		hFile := FilecontentManager.FileHandle,
		sNetId := FilecontentManager.AmsNetId,
		tTimeout := Timeout
	);	
END_IF

_Close(bExecute := TRUE);

IF _Close.bError THEN
	//exceptionFactory.ThrowException(__POSITION(), WStringHelper.Concat2("File close failed", GetErrorMessageByErrorId(_Close.nErrId)), _Close.nErrId);	
ELSIF NOT _Close.bBusy THEN
	FileContentManager.FilePath := '';
	FileContentManager.AmsNetId := '';
	FileContentManager.FileHandle := 0;

	Execute := EXECUTION_STATE.DONE;
END_IF
END_METHOD

END_FUNCTION_BLOCK

// ---- Files/FileContentManager/Tasks/FileFlushTask.TcPOU
{attribute 'enable_dynamic_creation'}	
{attribute 'no_explicit_call' := 'do not call this function block directly'} 
FUNCTION_BLOCK FileFlushTask EXTENDS FileContentTask
VAR
	_ClassName : STRING := __POUNAME();

	_Closed : BOOL;
	_Close : Tc2_System.FB_FileClose;
	_Open : Tc2_System.FB_FileOpen;
END_VAR

{attribute 'monitoring' := 'call'}
PROPERTY ClassName : STRING
GET
ClassName := _ClassName;
END_GET
END_PROPERTY

METHOD Execute : BOOL
VAR_INPUT
	start : BOOL;
END_VAR
VAR
	//exceptionFactory : ExceptionFactory(__POUNAME(), ClassName, CurrentNamespace.Name);
END_VAR
IF start THEN
	Validate();
	
	_Close(
		bExecute := FALSE,
		hFile := FileContentManager.FileHandle
	);
		
	_Open(
		bExecute := FALSE,
		sPathName := FileContentManager.FilePath,
		nMode := TO_DWORD(FileContentManager.OpenMode) OR TO_DWORD(FileContentManager.ContentHandlingMode),
		ePath := FileContentManager.PathType,
		sNetId := FilecontentManager.AmsNetId,
		tTimeout := Timeout
	);	
	
	_Closed := FALSE;	
END_IF

IF NOT _Closed THEN
	_Close(bExecute := TRUE);
	
	IF _Close.bError THEN
		//exceptionFactory.ThrowException(__POSITION(), WStringHelper.Concat2("File close for flush failed", GetErrorMessageByErrorId(_Close.nErrId)), _Close.nErrId);	
	ELSIF NOT _Close.bBusy THEN
		FileContentManager.FileHandle := 0;
		
		_Closed := TRUE;
	END_IF
END_IF
	
IF _Closed THEN
	_Open(bExecute := TRUE);
	
	IF _Open.bError THEN
		//exceptionFactory.ThrowException(__POSITION(), WStringHelper.Concat2("File open for flush failed", GetErrorMessageByErrorId(_Open.nErrId)), __POUNAME(), ClassName, CurrentNamespace.Name, __POSITION(), _Open.nErrId);	
	ELSIF NOT _Open.bBusy THEN
		FileContentManager.FileHandle := _Open.hFile;		
		
		Execute := EXECUTION_STATE.DONE;
	END_IF
END_IF
END_METHOD

END_FUNCTION_BLOCK

// ---- Files/FileContentManager/Tasks/FileGetCurrentPositionTask.TcPOU
{attribute 'enable_dynamic_creation'}	
{attribute 'no_explicit_call' := 'do not call this function block directly'} 
FUNCTION_BLOCK FileGetCurrentPositionTask EXTENDS FileContentTask
VAR
	_ClassName : STRING := __POUNAME();

    _GetCurrentPosition : Tc2_System.FB_FileTell;
END_VAR

{attribute 'monitoring' := 'call'}
PROPERTY ClassName : STRING
GET
ClassName := _ClassName;
END_GET
END_PROPERTY

METHOD Execute : BOOL
VAR_INPUT
	start : BOOL;
END_VAR
IF start THEN
	Validate();

	_GetCurrentPosition(
		bExecute := FALSE,
		hFile := FilecontentManager.FileHandle,
		sNetId := FilecontentManager.AmsNetId,
		tTimeout := Timeout
	);	
END_IF

_GetCurrentPosition(bExecute := TRUE);

IF _GetCurrentPosition.bError THEN
	//exceptionFactory.ThrowException(__POSITION(), WStringHelper.Concat2("Get current file position failed", GetErrorMessageByErrorId(_GetCurrentPosition.nErrId)), __POUNAME(), ClassName, CurrentNamespace.Name, __POSITION(), _GetCurrentPosition.nErrId);
ELSIF NOT _GetCurrentPosition.bBusy THEN
	Execute := EXECUTION_STATE.DONE;
END_IF
END_METHOD

PROPERTY FilePointerPosition : DINT
GET
FilePointerPosition := _GetCurrentPosition.nSeekPos;
END_GET
END_PROPERTY

END_FUNCTION_BLOCK

// ---- Files/FileContentManager/Tasks/FileMovePointerTask.TcPOU
{attribute 'enable_dynamic_creation'}	
{attribute 'no_explicit_call' := 'do not call this function block directly'} 
FUNCTION_BLOCK FileMovePointerTask EXTENDS FileContentTask
VAR
	_ClassName : STRING := __POUNAME();

    _MovePointer : Tc2_System.FB_FileSeek;
END_VAR

{attribute 'monitoring' := 'call'}
PROPERTY ClassName : STRING
GET
ClassName := _ClassName;
END_GET
END_PROPERTY

METHOD Execute : BOOL
VAR_INPUT
	start : BOOL;
END_VAR
IF start THEN
	Validate();

	_MovePointer(
		bExecute := FALSE,
		hFile := FilecontentManager.FileHandle,
		sNetId := FilecontentManager.AmsNetId,
		tTimeout := Timeout
	);	
END_IF

_MovePointer(bExecute := TRUE);

IF _MovePointer.bError THEN
	//exceptionFactory.ThrowException(__POSITION(), WStringHelper.Concat2("Move file pointer failed", GetErrorMessageByErrorId(_MovePointer.nErrId)), __POUNAME(), ClassName, CurrentNamespace.Name, __POSITION(), _MovePointer.nErrId);
ELSIF NOT _MovePointer.bBusy THEN
	Execute := EXECUTION_STATE.DONE;
END_IF
END_METHOD

PROPERTY MovePointerType : FILE_MOVE_POINTER_TYPE
GET
VAR
	resultAddress : POINTER TO INT;
END_VAR
resultAddress := ADR(MovePointerType);
resultAddress^ := _MovePointer.eOrigin;
END_GET
SET
_MovePointer.eOrigin := TO_INT(MovePointerType);
END_SET
END_PROPERTY

PROPERTY NewFilePointerPosition : DINT
GET
NewFilePointerPosition := _MovePointer.nSeekPos;
END_GET
SET
_MovePointer.nSeekPos := NewFilePointerPosition;
END_SET
END_PROPERTY

END_FUNCTION_BLOCK

// ---- Files/FileContentManager/Tasks/FileOpenTask.TcPOU
{attribute 'enable_dynamic_creation'}	
{attribute 'no_explicit_call' := 'do not call this function block directly'} 
FUNCTION_BLOCK FileOpenTask EXTENDS FileContentTask
VAR
	_ClassName : STRING := __POUNAME();

	_Open : Tc2_System.FB_FileOpen;
	_OpenMode : FILE_OPEN_MODE;
	_ContentHandlingMode : FILE_CONTENT_HANDLING_MODE;		
END_VAR

{attribute 'monitoring' := 'call'}
{attribute 'OPC.UA.DA.Property' := '1'}
PROPERTY AmsNetId : Tc2_System.T_AmsNetID
GET
AmsNetId := _Open.sNetId;
END_GET
SET
_Open.sNetId := AmsNetId;
END_SET
END_PROPERTY

{attribute 'monitoring' := 'call'}
PROPERTY ClassName : STRING
GET
ClassName := _ClassName;
END_GET
END_PROPERTY

{attribute 'monitoring' := 'call'}
{attribute 'OPC.UA.DA.Property' := '1'}
PROPERTY ContentHandlingMode : FILE_CONTENT_HANDLING_MODE
GET
ContentHandlingMode := _ContentHandlingMode;
END_GET
SET
_ContentHandlingMode := ContentHandlingMode;
END_SET
END_PROPERTY

METHOD Execute : BOOL
VAR_INPUT
	start : BOOL;
END_VAR
VAR
	
END_VAR
IF start THEN
	Validate();
	
	_Open(
		bExecute := FALSE,
		nMode := TO_DWORD(openMode) OR TO_DWORD(contentHandlingMode),
		tTimeout := Timeout 
	);	
END_IF

_Open(bExecute := TRUE);

IF _Open.bError THEN
	//exceptionFactory.ThrowException(__POSITION(), WStringHelper.Concat2("File open failed", GetErrorMessageByErrorId(_Open.nErrId)), __POUNAME(), ClassName, CurrentNamespace.Name, __POSITION(), _Open.nErrId);	
ELSIF NOT _Open.bBusy THEN
	FileContentManager.FilePath := _Open.sPathName;
	FileContentManager.OpenMode := _OpenMode;
	FileContentManager.ContentHandlingMode := _ContentHandlingMode;
	FileContentManager.PathType := _Open.ePath;
	FileContentManager.AmsNetId := _Open.sNetId;
	FileContentManager.FileHandle := _Open.hFile;
	
	Execute := EXECUTION_STATE.DONE;
END_IF
END_METHOD

{attribute 'monitoring' := 'call'}
{attribute 'OPC.UA.DA.Property' := '1'}
PROPERTY FilePath : Tc2_System.T_MaxString
GET
FilePath := _Open.sPathName;
END_GET
SET
_Open.sPathName := FilePath;
END_SET
END_PROPERTY

{attribute 'monitoring' := 'call'}
{attribute 'OPC.UA.DA.Property' := '1'}
PROPERTY OpenMode : FILE_OPEN_MODE
GET
OpenMode := _OpenMode;
END_GET
SET
_OpenMode := OpenMode;
END_SET
END_PROPERTY

{attribute 'monitoring' := 'call'}
{attribute 'OPC.UA.DA.Property' := '1'}
{attribute 'OPC.UA.DA.Access' := '1'}
PROPERTY PathType : E_OpenPath
GET
PathType := _Open.ePath;
END_GET
SET
_Open.ePath := PathType;
END_SET
END_PROPERTY

METHOD PROTECTED Validate
IF NOT __ISVALIDREF(FileContentManager) THEN
	//exceptionFactory.ThrowException(__POSITION(), "File content menager is not specified");
END_IF

IF FilePath = '' THEN
	//exceptionFactory.ThrowException(__POSITION(), "File path is not specified");
END_IF
END_METHOD

END_FUNCTION_BLOCK

// ---- Files/FileContentManager/Tasks/FileReadBytesTask.TcPOU
{attribute 'enable_dynamic_creation'}	
{attribute 'no_explicit_call' := 'do not call this function block directly'} 
FUNCTION_BLOCK FileReadBytesTask EXTENDS FileContentTask
VAR
	_ClassName : STRING := __POUNAME();

	_ReadBytes : Tc2_System.FB_FileRead;
	_TargetBuffer : DynamicByteArray;
END_VAR

{attribute 'monitoring' := 'call'}
PROPERTY ClassName : STRING
GET
ClassName := _ClassName;
END_GET
END_PROPERTY

METHOD Execute : BOOL
VAR_INPUT
	start : BOOL;
END_VAR
IF start THEN
	Validate();

	_ReadBytes(		
		bExecute := FALSE,
		hFile := FilecontentManager.FileHandle,
		pReadBuff := _TargetBuffer.Address,
		cbReadLen := MaxBytesToReadCount,
		sNetId := FilecontentManager.AmsNetId,
		tTimeout := Timeout
	);	
END_IF

_ReadBytes(bExecute := TRUE);

IF _ReadBytes.bError THEN
	//exceptionFactory.ThrowException(__POSITION(), WStringHelper.Concat2("Read string to file failed", GetErrorMessageByErrorId(_ReadBytes.nErrId)), __POUNAME(), ClassName, CurrentNamespace.Name, __POSITION(), _ReadBytes.nErrId);
ELSIF NOT _ReadBytes.bBusy THEN
	Execute := EXECUTION_STATE.DONE;
END_IF
END_METHOD

PROPERTY LoadedBytes : POINTER TO BYTE
GET
LoadedBytes := _TargetBuffer.Address;
END_GET
END_PROPERTY

PROPERTY LoadedBytesCount : UDINT
GET
LoadedBytesCount := _ReadBytes.cbRead;
END_GET
END_PROPERTY

PROPERTY MaxBytesToReadCount : UDINT
GET
MaxBytesToReadCount := TO_UDINT(_TargetBuffer.Count);
END_GET
SET
_TargetBuffer.Resize(TO_DINT(MaxBytesToReadCount));
END_SET
END_PROPERTY

METHOD PROTECTED Validate
SUPER^.Validate();

CASE FileContentManager.OpenMode OF
	FILE_OPEN_MODE.APPEND, FILE_OPEN_MODE.WRITE_EMPTY:
		//exceptionFactory.ThrowException(__POSITION(), "File is not open for reading");
END_CASE

IF FileContentManager.ContentHandlingMode <> FILE_CONTENT_HANDLING_MODE.BINARY THEN
	//exceptionFactory.ThrowException(__POSITION(), "File is not open in binary mode");
END_IF

IF _TargetBuffer.Count < 1 THEN
	//exceptionFactory.ThrowException(__POSITION(), "Buffer is empty (MaxBytesToReadCount has value 0)");
END_IF
END_METHOD

END_FUNCTION_BLOCK

// ---- Files/FileContentManager/Tasks/FileReadStringTask.TcPOU
{attribute 'enable_dynamic_creation'}	
{attribute 'no_explicit_call' := 'do not call this function block directly'} 
FUNCTION_BLOCK FileReadStringTask EXTENDS FileContentTask
VAR
	_ClassName : STRING := __POUNAME();

	_ReadString : Tc2_System.FB_FileGets;
END_VAR

{attribute 'monitoring' := 'call'}
PROPERTY ClassName : STRING
GET
ClassName := _ClassName;
END_GET
END_PROPERTY

METHOD Execute : BOOL
VAR_INPUT
	start : BOOL;
END_VAR
IF start THEN
	Validate();

	_ReadString(
		bExecute := FALSE,
		hFile := FilecontentManager.FileHandle,
		sNetId := FilecontentManager.AmsNetId,
		tTimeout := Timeout
	);	
END_IF

_ReadString(bExecute := TRUE);

IF _ReadString.bError THEN
	//exceptionFactory.ThrowException(__POSITION(), WStringHelper.Concat2("Read string from file failed", GetErrorMessageByErrorId(_ReadString.nErrId)), __POUNAME(), ClassName, CurrentNamespace.Name, __POSITION(), _ReadString.nErrId);
ELSIF NOT _ReadString.bBusy THEN
	Execute := EXECUTION_STATE.DONE;
END_IF
END_METHOD

PROPERTY LoadedString : REFERENCE TO Tc2_System.T_MaxString
GET
LoadedString REF= _ReadString.sLine;
END_GET
END_PROPERTY

METHOD PROTECTED Validate
SUPER^.Validate();

CASE FileContentManager.OpenMode OF
	FILE_OPEN_MODE.APPEND, FILE_OPEN_MODE.WRITE_EMPTY:
		//exceptionFactory.ThrowException(__POSITION(), "File is not open for reading");
END_CASE

IF FileContentManager.ContentHandlingMode <> FILE_CONTENT_HANDLING_MODE.TEXT THEN
	//exceptionFactory.ThrowException(__POSITION(), "File is not open in text mode");
END_IF
END_METHOD

END_FUNCTION_BLOCK

// ---- Files/FileContentManager/Tasks/FileTestForEndTask.TcPOU
{attribute 'enable_dynamic_creation'}	
{attribute 'no_explicit_call' := 'do not call this function block directly'} 
FUNCTION_BLOCK FileTestForEndTask EXTENDS FileContentTask
VAR
	_ClassName : STRING := __POUNAME();

	_TestForEndOfFile : Tc2_System.FB_EOF;
END_VAR

{attribute 'monitoring' := 'call'}
PROPERTY ClassName : STRING
GET
ClassName := _ClassName;
END_GET
END_PROPERTY

METHOD Execute : BOOL
VAR_INPUT
	start : BOOL;
END_VAR
IF start THEN
	Validate();

	_TestForEndOfFile(
		bExecute := FALSE,
		hFile := FilecontentManager.FileHandle,
		sNetId := FilecontentManager.AmsNetId,
		tTimeout := Timeout
	);	
END_IF

_TestForEndOfFile(bExecute := TRUE);

IF _TestForEndOfFile.bError THEN
	//exceptionFactory.ThrowException(__POSITION(), WStringHelper.Concat2("Test for end of file failed", GetErrorMessageByErrorId(_TestForEndOfFile.nErrId)), __POUNAME(), ClassName, CurrentNamespace.Name, __POSITION(), _TestForEndOfFile.nErrId);
ELSIF NOT _TestForEndOfFile.bBusy THEN
	Execute := EXECUTION_STATE.DONE;
END_IF
END_METHOD

PROPERTY IsEndOffile : BOOL
GET
IsEndOffile := _TestForEndOfFile.bEOF;
END_GET
END_PROPERTY

END_FUNCTION_BLOCK

// ---- Files/FileContentManager/Tasks/FileWriteBytesTask.TcPOU
{attribute 'enable_dynamic_creation'}	
{attribute 'no_explicit_call' := 'do not call this function block directly'} 
FUNCTION_BLOCK FileWriteBytesTask EXTENDS FileContentTask
VAR
	_ClassName : STRING := __POUNAME();

    _WriteBytes : Tc2_System.FB_FileWrite;
	_SourceBuffer : DynamicByteArray;
END_VAR

PROPERTY BytesToWrite : REFERENCE TO DynamicByteArray
GET
BytesToWrite REF= _SourceBuffer;
END_GET
END_PROPERTY

{attribute 'monitoring' := 'call'}
PROPERTY ClassName : STRING
GET
ClassName := _ClassName;
END_GET
END_PROPERTY

METHOD Execute : BOOL
VAR_INPUT
	start : BOOL;
END_VAR
IF start THEN
	Validate();

	_WriteBytes(
		bExecute := FALSE,
		hFile := FilecontentManager.FileHandle,
		pWriteBuff := _SourceBuffer.Address,
		cbWriteLen := TO_UDINT(_SourceBuffer.Count),
		sNetId := FilecontentManager.AmsNetId,
		tTimeout := Timeout 
	);	
END_IF

_WriteBytes(bExecute := TRUE);

IF _WriteBytes.bError THEN
	//exceptionFactory.ThrowException(__POSITION(), WStringHelper.Concat2("Write bytes to file failed", GetErrorMessageByErrorId(_WriteBytes.nErrId)), __POUNAME(), ClassName, CurrentNamespace.Name, __POSITION(), _WriteBytes.nErrId);
ELSIF NOT _WriteBytes.bBusy THEN
	Execute := EXECUTION_STATE.DONE;
END_IF
END_METHOD

METHOD PROTECTED Validate
SUPER^.Validate();

CASE FileContentManager.OpenMode OF
	FILE_OPEN_MODE.READ_EXISTING:
		//exceptionFactory.ThrowException(__POSITION(), "File is not open for writing");
END_CASE

IF FileContentManager.ContentHandlingMode <> FILE_CONTENT_HANDLING_MODE.BINARY THEN
	//exceptionFactory.ThrowException(__POSITION(), "File is not open in binary mode");
END_IF
END_METHOD

PROPERTY WrittenBytesCount : UDINT
GET
WrittenBytesCount := _WriteBytes.cbWrite;
END_GET
END_PROPERTY

END_FUNCTION_BLOCK

// ---- Files/FileContentManager/Tasks/FileWriteStringTask.TcPOU
{attribute 'enable_dynamic_creation'}	
{attribute 'no_explicit_call' := 'do not call this function block directly'} 
FUNCTION_BLOCK FileWriteStringTask EXTENDS FileContentTask
VAR
	_ClassName : STRING := __POUNAME();

	_WriteString : Tc2_System.FB_FilePuts;
END_VAR

{attribute 'monitoring' := 'call'}
PROPERTY ClassName : STRING
GET
ClassName := _ClassName;
END_GET
END_PROPERTY

METHOD Execute : BOOL
VAR_INPUT
	start : BOOL;
END_VAR
IF start THEN
	Validate();

	_WriteString(
		bExecute := FALSE,
		hFile := FilecontentManager.FileHandle,
		sNetId := FilecontentManager.AmsNetId,
		tTimeout := Timeout
	); 
END_IF

_WriteString(bExecute := TRUE);

IF _WriteString.bError THEN
	//exceptionFactory.ThrowException(__POSITION(), WStringHelper.Concat2("Write string to file failed", GetErrorMessageByErrorId(_WriteString.nErrId)), __POUNAME(), ClassName, CurrentNamespace.Name, __POSITION(), _WriteString.nErrId);
ELSIF NOT _WriteString.bBusy THEN
	Execute := EXECUTION_STATE.DONE;
END_IF
END_METHOD

PROPERTY StringToWrite : REFERENCE TO Tc2_System.T_MaxString
GET
StringToWrite REF= _WriteString.sLine;
END_GET
END_PROPERTY

METHOD PROTECTED Validate
SUPER^.Validate();

CASE FileContentManager.OpenMode OF
	FILE_OPEN_MODE.READ_EXISTING:
		//exceptionFactory.ThrowException(__POSITION(), "File is not open for writing");
END_CASE

IF FileContentManager.ContentHandlingMode <> FILE_CONTENT_HANDLING_MODE.TEXT THEN
	//exceptionFactory.ThrowException(__POSITION(), "File is not open in text mode");
END_IF
END_METHOD

END_FUNCTION_BLOCK

// ---- Files/LoadFile.TcPOU
{attribute 'no_explicit_call' := 'do not call this function block directly'} 
FUNCTION_BLOCK LoadFile EXTENDS ToolkitObject IMPLEMENTS IAction
VAR
	{attribute 'OPC.UA.DA' := '0'}
	_ClassName : STRING := __POUNAME();

	{attribute 'OPC.UA.DA' := '0'}
    _Load : Tc2_System.FB_FileLoad; 
	
	{attribute 'OPC.UA.DA' := '0'}
	_NeedStart : BOOL;
	{attribute 'OPC.UA.DA' := '0'}
	_Done : BOOL;
END_VAR

{attribute 'monitoring' := 'call'}
{attribute 'OPC.UA.DA.Property' := '1'}
{attribute 'OPC.UA.DA' := '1'}
PROPERTY AmsNetId : Tc2_System.T_AmsNetID
GET
AmsNetId := _Load.sNetId;
END_GET
SET
_Load.sNetId := AmsNetId;
END_SET
END_PROPERTY

{attribute 'monitoring' := 'call'}
{attribute 'OPC.UA.DA.Property' := '1'}
{attribute 'OPC.UA.DA.Access' := '1'}
PROPERTY Busy : BOOL
GET
Busy := _NeedStart OR_ELSE _Load.bBusy;
END_GET
END_PROPERTY

{attribute 'monitoring' := 'call'}
PROPERTY ClassName : STRING
GET
ClassName := _ClassName;
END_GET
END_PROPERTY

{attribute 'monitoring' := 'call'}
{attribute 'OPC.UA.DA.Property' := '1'}
{attribute 'OPC.UA.DA.Access' := '1'}
PROPERTY Done : BOOL
GET
Done := _Done;
END_GET
END_PROPERTY

{attribute 'monitoring' := 'call'}
{attribute 'OPC.UA.DA.Property' := '1'}
{attribute 'OPC.UA.DA.Access' := '1'}
PROPERTY Error : BOOL
GET
Error := _Load.bError;
END_GET
END_PROPERTY

METHOD Execute
VAR
	message : ERROR_MESSAGE;
END_VAR
IF _NeedStart OR_ELSE _Load.bBusy THEN
	_Load(bExecute := TRUE);
	_NeedStart := FALSE;
	
	IF _Load.bError THEN
		message := "An error occurred while loading the file '";
		WStringHelper.Append2(message, TO_WSTRING(_Load.sPathName), "'");	
		_LastException.Configure(message, __POUNAME(), ClassName, CurrentNamespace.Name, __POSITION(), _Load.nErrId).Throw();
	ELSIF NOT _Load.bBusy THEN
		_Done := TRUE;
	END_IF
END_IF
END_METHOD

{attribute 'monitoring' := 'call'}
{attribute 'OPC.UA.DA.Property' := '1'}
{attribute 'OPC.UA.DA.Access' := '1'}
PROPERTY LastException : REFERENCE TO Exception
GET
LastException REF= _LastException;
END_GET
END_PROPERTY

METHOD Start
VAR_INPUT
	filePath : Tc2_System.T_MaxString;
	targetBuffer : __System.AnyType;
END_VAR
_NeedStart := TRUE;
_Done := FALSE;
_Load.sPathName := filePath;
_Load.pReadBuff := targetBuffer.pValue;
_Load.cbReadLen := TO_UDINT(targetBuffer.diSize);

_LastException.Clear();
END_METHOD

{attribute 'monitoring' := 'call'}
{attribute 'OPC.UA.DA.Property' := '1'}
{attribute 'OPC.UA.DA' := '1'}
PROPERTY Timeout : TIME
GET
Timeout := _Load.tTimeout;
END_GET
SET
_Load.tTimeout := Timeout;
END_SET
END_PROPERTY

END_FUNCTION_BLOCK

// ---- Files/RenameFile.TcPOU
{attribute 'no_explicit_call' := 'do not call this function block directly'} 
FUNCTION_BLOCK RenameFile EXTENDS ToolkitObject IMPLEMENTS IAction
VAR
	{attribute 'OPC.UA.DA' := '0'}
	_ClassName : STRING := __POUNAME();

	{attribute 'OPC.UA.DA' := '0'}
    _Rename : Tc2_System.FB_FileRename;
	
	{attribute 'OPC.UA.DA' := '0'}
	_NeedStart : BOOL;
	{attribute 'OPC.UA.DA' := '0'}
	_Done : BOOL;
END_VAR

{attribute 'monitoring' := 'call'}
{attribute 'OPC.UA.DA.Property' := '1'}
{attribute 'OPC.UA.DA' := '1'}
PROPERTY AmsNetId : Tc2_System.T_AmsNetID
GET
AmsNetId := _Rename.sNetId;
END_GET
SET
_Rename.sNetId := AmsNetId;
END_SET
END_PROPERTY

{attribute 'monitoring' := 'call'}
{attribute 'OPC.UA.DA.Property' := '1'}
{attribute 'OPC.UA.DA.Access' := '1'}
PROPERTY Busy : BOOL
GET
Busy := _NeedStart OR_ELSE _Rename.bBusy;
END_GET
END_PROPERTY

{attribute 'monitoring' := 'call'}
PROPERTY ClassName : STRING
GET
ClassName := _ClassName;
END_GET
END_PROPERTY

{attribute 'monitoring' := 'call'}
{attribute 'OPC.UA.DA.Property' := '1'}
{attribute 'OPC.UA.DA.Access' := '1'}
PROPERTY Done : BOOL
GET
Done := _Done;
END_GET
END_PROPERTY

{attribute 'monitoring' := 'call'}
{attribute 'OPC.UA.DA.Property' := '1'}
{attribute 'OPC.UA.DA.Access' := '1'}
PROPERTY Error : BOOL
GET
Error := _Rename.bError;
END_GET
END_PROPERTY

METHOD Execute
VAR
	message : ERROR_MESSAGE;
END_VAR
IF _NeedStart OR_ELSE _Rename.bBusy THEN
	_Rename(bExecute := TRUE);
	_NeedStart := FALSE;
	
	IF _Rename.bError THEN
		message := "An error occurred while renaming the file '";
		WStringHelper.Append6(message, TO_WSTRING(_Rename.sOldName), "' to '", TO_WSTRING(_Rename.sNewName), " in directory '", TO_WSTRING(_Rename.ePath), "'");	
		_LastException.Configure(message, __POUNAME(), ClassName, CurrentNamespace.Name, __POSITION(), _Rename.nErrId);
	ELSIF NOT _Rename.bBusy THEN
		_Done := TRUE;
	END_IF
END_IF
END_METHOD

{attribute 'monitoring' := 'call'}
{attribute 'OPC.UA.DA.Property' := '1'}
{attribute 'OPC.UA.DA.Access' := '1'}
PROPERTY LastException : REFERENCE TO Exception
GET
LastException REF= _LastException;
END_GET
END_PROPERTY

{attribute 'monitoring' := 'call'}
{attribute 'OPC.UA.DA.Property' := '1'}
{attribute 'OPC.UA.DA' := '1'}
PROPERTY PathType : Tc2_System.E_OpenPath
GET
PathType := _Rename.ePath;
END_GET
SET
_Rename.ePath := PathType;
END_SET
END_PROPERTY

METHOD Start
VAR_INPUT
	oldFilePath : Tc2_System.T_MaxString;
	newFilePath : Tc2_System.T_MaxString;
END_VAR
_NeedStart := TRUE;
_Done := FALSE;
_Rename.sOldName := oldFilePath;
_Rename.sNewName := newFilePath;

_LastException.Clear();
END_METHOD

{attribute 'monitoring' := 'call'}
{attribute 'OPC.UA.DA.Property' := '1'}
{attribute 'OPC.UA.DA' := '1'}
PROPERTY Timeout : TIME
GET
Timeout := _Rename.tTimeout;
END_GET
SET
_Rename.tTimeout := Timeout;
END_SET
END_PROPERTY

END_FUNCTION_BLOCK

// ---- StateMachine/Finite/FiniteStateMachine.TcPOU
{attribute 'no_explicit_call' := 'do not call this function block directly'} 
FUNCTION_BLOCK ABSTRACT FiniteStateMachine EXTENDS ToolkitObject
VAR_INPUT
	{attribute 'OPC.UA.DA' := '0'}
	RequestedCause : STRING;	

	{attribute 'OPC.UA.DA.Access' := '1'}
	CurrentState : REFERENCE TO ProgramState;
	
	{attribute 'OPC.UA.DA.Access' := '1'}
	LastTransition : REFERENCE TO ProgramTransition;
END_VAR
VAR	
	{attribute 'OPC.UA.DA' := '0'}
	_AvailableStates : ARRAY [0..ProgramConstants.MaxStateCount - 1] OF POINTER TO ProgramState;

	{attribute 'OPC.UA.DA' := '0'}
	_AvailableTransitions : ARRAY [0..ProgramConstants.MaxTransitionCount - 1] OF POINTER TO ProgramTransition;
END_VAR

{attribute 'monitoring' := 'call'}
{attribute 'OPC.UA.DA.Property' := '1'}
{attribute 'OPC.UA.DA.Access' := '1'}
PROPERTY ABSTRACT AvailableStateCount : INT(0..ProgramConstants.MaxStateCount - 1)
GET
END_GET
END_PROPERTY

{attribute 'monitoring' := 'call'}
{attribute 'OPC.UA.DA.Property' := '1'}
{attribute 'OPC.UA.DA.Access' := '1'}
PROPERTY ABSTRACT AvailableTransitionCount : INT(0..ProgramConstants.MaxTransitionCount - 1)
GET
END_GET
END_PROPERTY

METHOD INTERNAL Clear
CurrentState REF= 0;
LastTransition REF= 0;

LastException.Clear();
END_METHOD

{attribute 'monitoring' := 'call'}
PROPERTY CurrentStateName : STRING
GET
IF __ISVALIDREF(CurrentState) THEN
	CurrentStateName := CurrentState.Name;
END_IF
END_GET
END_PROPERTY

METHOD Execute
VAR
	newState : POINTER TO ProgramState;
	newTransition : POINTER TO ProgramTransition;
END_VAR
(*IF InTransition THEN
	LastTransition.Execute();
		
	IF LastTransition.Error THEN
		LastException := LastTransition.LastException;
		exceptionSet.AddExisting(LastException);
		RETURN;
	ELSIF LastTransition.Busy THEN
		Execute := TRUE;
		RETURN;
	ELSIF LastTransition.Done THEN
		IF newState := GetStateByName(LastTransition.ToState) THEN
			CurrentState REF= newState^;			
			CurrentState.Enable();
			
			IF CurrentState.Error THEN				
				LastException := CurrentState.LastException;
				exceptionSet.AddExisting(LastException);
				RETURN;
			END_IF
		ELSE
			exceptionSet.AddExisting(LastException);
			RETURN;
		END_IF
	ELSE
		Last//exceptionFactory.ThrowException(__POSITION(), 0, WStringHelper.Concat3("CurrentTransition ", TO_WSTRING(LastTransition.Name), " is not in busy, done or error state"));
		exceptionSet.AddExisting(LastException);
		RETURN;		
	END_IF
END_IF

IF NOT __ISVALIDREF(CurrentState) THEN
	Last//exceptionFactory.ThrowException(__POSITION(), 0, "CurrentState is null");
	exceptionSet.AddExisting(LastException);
	RETURN;
END_IF

IF RequestedCause <> '' THEN
	IF FindTransitionByCause(RequestedCause, transition => newTransition, exception => LastException) THEN
		RequestedCause := '';
		
		IF CurrentState.Busy THEN
			CurrentState.Disable();			
		END_IF
		
		LastTransition REF= newTransition^;
		LastTransition.Start();

		IF NOT LastTransition.Error THEN
			Execute := TRUE;
		ELSE				
			LastException := LastTransition.LastException;
			exceptionSet.AddExisting(LastException);
		END_IF
		
		RETURN;		
	ELSE
		RequestedCause := '';
		exceptionSet.AddExisting(LastException);
		RETURN;
	END_IF
END_IF

IF CurrentState.Busy THEN 
	CurrentState.Execute();
	
	IF CurrentState.Error THEN
		LastException := CurrentState.LastException;
		exceptionSet.AddExisting(LastException);
		RETURN;
	ELSIF NOT CurrentState.Busy THEN
		Last//exceptionFactory.ThrowException(__POSITION(), 0, WStringHelper.Concat3("CurrentState ", TO_WSTRING(CurrentState.Name), " is not in busy or error state"));
		exceptionSet.AddExisting(LastException);
		RETURN;		
	END_IF
END_IF

Execute := TRUE;*)
END_METHOD

METHOD PROTECTED FINAL FindTransitionByCause : POINTER TO ProgramTransition
VAR_INPUT
	cause : STRING;
END_VAR
VAR
	i : INT;
END_VAR
IF NOT __ISVALIDREF(CurrentState) THEN
	//exceptionFactory.ThrowException(__POSITION(), WStringHelper.Concat4("Unsupported cause ", TO_WSTRING(cause), " to make transition from state ", TO_WSTRING(CurrentState.Name)));
END_IF

FOR i := 0 TO AvailableTransitionCount - 1 DO
	IF _AvailableTransitions[i]^.FromState = CurrentState.Name AND_THEN _AvailableTransitions[i]^.Cause = cause THEN
		FindTransitionByCause := _AvailableTransitions[i];
		RETURN;
	END_IF
END_FOR

//exceptionFactory.ThrowException(__POSITION(), WStringHelper.Concat4("Unsupported cause ", TO_WSTRING(cause), " to make transition from state ", TO_WSTRING(CurrentState.Name)));
END_METHOD

METHOD PROTECTED FINAL GetStateByName : POINTER TO ProgramState
VAR_INPUT
	name : STRING;
END_VAR
VAR
	i : INT;
END_VAR
FOR i := 0 TO AvailableStateCount - 1 DO
	IF _AvailableStates[i]^.Name = name THEN
		GetStateByName := _AvailableStates[i];
		RETURN;
	END_IF
END_FOR

//exceptionFactory.ThrowException(__POSITION(), WStringHelper.Concat2("Unknown state with name ", TO_WSTRING(name)));
END_METHOD

METHOD Initialize 
VAR
	i, j : INT;
	defaultState : POINTER TO ProgramState;
END_VAR
InternalInitialize(states => _AvailableStates, transitions => _AvailableTransitions, defaultState => defaultState);

IF AvailableStateCount <= 0 OR_ELSE AvailableStateCount > ProgramConstants.MaxStateCount - 1 THEN
	//exceptionFactory.ThrowException(__POSITION(), WStringHelper.Concat2("Invalid state count  ", TO_WSTRING(AvailableStateCount)));
END_IF

IF AvailableTransitionCount <= 0 OR_ELSE AvailableTransitionCount > ProgramConstants.MaxTransitionCount - 1 THEN
	//exceptionFactory.ThrowException(__POSITION(), WStringHelper.Concat2("Invalid transition count  ", TO_WSTRING(AvailableTransitionCount)));
END_IF

IF defaultState = 0 THEN
	//exceptionFactory.ThrowException(__POSITION(), "Default state is not specified");
END_IF

FOR i := 0 TO AvailableStateCount - 1 DO
	FOR j := 0 TO AvailableTransitionCount - 1 DO
		IF _AvailableStates[i]^.Name = _AvailableTransitions[j]^.FromState OR_ELSE _AvailableStates[i]^.Name = _AvailableTransitions[j]^.ToState THEN
			_AvailableStates[i]^.RegisterTransition(_AvailableTransitions[j]^);
		END_IF
	END_FOR	
END_FOR

CurrentState REF= defaultState^;
END_METHOD

METHOD PROTECTED ABSTRACT InternalInitialize 
VAR_OUTPUT
	states : ARRAY [0..ProgramConstants.MaxStateCount - 1] OF POINTER TO ProgramState;
	transitions : ARRAY [0..ProgramConstants.MaxTransitionCount - 1] OF POINTER TO ProgramTransition;
	defaultState : POINTER TO ProgramState;
END_VAR
END_METHOD

{attribute 'monitoring' := 'call'}
{attribute 'OPC.UA.DA.Property' := '1'}
{attribute 'OPC.UA.DA.Access' := '1'}
PROPERTY InTransition : BOOL
GET
InTransition := __ISVALIDREF(LastTransition) AND_THEN LastTransition.Busy;
END_GET
END_PROPERTY

{attribute 'monitoring' := 'call'}
PROPERTY LastTransitionName : STRING
GET
IF __ISVALIDREF(LastTransition) THEN
	LastTransitionName := LastTransition.Name;
END_IF
END_GET
END_PROPERTY

END_FUNCTION_BLOCK

// ---- StateMachine/Finite/ProgramState.TcPOU
{attribute 'no_explicit_call' := 'do not call this function block directly'} 
FUNCTION_BLOCK ABSTRACT ProgramState EXTENDS ToolkitObject
VAR_OUTPUT
	{attribute 'OPC.UA.DA.Access' := '1'}
	FromTransitions : ARRAY [0..ProgramConstants.MaxTransitionCount - 1] OF STRING;
	{attribute 'OPC.UA.DA.Access' := '1'}
	FromTransitionCount : INT(0..ProgramConstants.MaxTransitionCount - 1);
	{attribute 'OPC.UA.DA.Access' := '1'}
	ToTransitions : ARRAY [0..ProgramConstants.MaxTransitionCount - 1] OF STRING;
	{attribute 'OPC.UA.DA.Access' := '1'}
	ToTransitionCount : INT(0..ProgramConstants.MaxTransitionCount - 1);
END_VAR
VAR
	{attribute 'OPC.UA.DA' := '0'}
	_Busy : BOOL;
	{attribute 'OPC.UA.DA' := '0'}
	_Error : BOOL;

	{attribute 'OPC.UA.DA' := '0'}
	_StateMachine : REFERENCE TO FiniteStateMachine;
END_VAR

{attribute 'monitoring' := 'call'}
{attribute 'OPC.UA.DA.Property' := '1'}
{attribute 'OPC.UA.DA.Access' := '1'}
PROPERTY Busy : BOOL
GET
Busy := _Busy;
END_GET
END_PROPERTY

METHOD Disable
IF _Busy THEN
	_Busy := FALSE;
END_IF
END_METHOD

METHOD Enable
_Busy := TRUE;
_Error := FALSE;
END_METHOD

{attribute 'monitoring' := 'call'}
{attribute 'OPC.UA.DA.Property' := '1'}
{attribute 'OPC.UA.DA.Access' := '1'}
PROPERTY Error : BOOL
GET
Error := _Error;
END_GET
END_PROPERTY

METHOD Execute
END_METHOD

METHOD Initialize 
VAR_INPUT
	stateMachine : REFERENCE TO FiniteStateMachine;
END_VAR
IF NOT __ISVALIDREF(_StateMachine) THEN
	//exceptionFactory.ThrowException(__POSITION(), "programStateMachine is NULL");
END_IF

_StateMachine REF= stateMachine;
END_METHOD

{attribute 'monitoring' := 'call'}
{attribute 'OPC.UA.DA.Property' := '1'}
{attribute 'OPC.UA.DA.Access' := '1'}
PROPERTY Initialized : BOOL
GET
Initialized := __ISVALIDREF(_StateMachine);
END_GET
END_PROPERTY

{attribute 'monitoring' := 'call'}
PROPERTY LastException : REFERENCE TO Exception
GET
LastException REF= _LastException;
END_GET
END_PROPERTY

{attribute 'monitoring' := 'call'}
{attribute 'OPC.UA.DA.Property' := '1'}
{attribute 'OPC.UA.DA.Access' := '1'}
PROPERTY ABSTRACT Name : STRING
GET
END_GET
END_PROPERTY

METHOD INTERNAL FINAL RegisterTransition
VAR_INPUT
	transition : REFERENCE TO ProgramTransition;
END_VAR
IF transition.FromState = Name THEN
	ToTransitions[ToTransitionCount] := transition.Name;
	ToTransitionCount := ToTransitionCount + 1;
ELSIF transition.ToState = Name THEN
	FromTransitions[FromTransitionCount] := transition.Name;
	FromTransitionCount := FromTransitionCount + 1;
END_IF
END_METHOD

END_FUNCTION_BLOCK

// ---- StateMachine/Finite/ProgramTransition.TcPOU
{attribute 'no_explicit_call' := 'do not call this function block directly'} 
FUNCTION_BLOCK ABSTRACT ProgramTransition EXTENDS ToolkitObject IMPLEMENTS IAction
VAR_OUTPUT
	//{attribute 'OPC.UA.DA.Access' := '1'}
	//Timeout : TIME := T#3S;
END_VAR
VAR
	{attribute 'OPC.UA.DA' := '0'}
	_Busy : BOOL;
	{attribute 'OPC.UA.DA' := '0'}
	_Done : BOOL;
	{attribute 'OPC.UA.DA' := '0'}
	_Error : BOOL;
	{attribute 'OPC.UA.DA' := '0'}
	_StateMachine : REFERENCE TO FiniteStateMachine;
END_VAR

{attribute 'monitoring' := 'call'}
{attribute 'OPC.UA.DA.Property' := '1'}
{attribute 'OPC.UA.DA.Access' := '1'}
PROPERTY Busy : BOOL
GET
Busy := _Busy;
END_GET
END_PROPERTY

METHOD Cancel
IF _Busy THEN
	_Busy := FALSE;	
END_IF
END_METHOD

{attribute 'monitoring' := 'call'}
{attribute 'OPC.UA.DA.Property' := '1'}
{attribute 'OPC.UA.DA.Access' := '1'}
PROPERTY ABSTRACT Cause : STRING
GET
END_GET
END_PROPERTY

{attribute 'monitoring' := 'call'}
{attribute 'OPC.UA.DA.Property' := '1'}
{attribute 'OPC.UA.DA.Access' := '1'}
PROPERTY Done : BOOL
GET
Done := _Done;
END_GET
END_PROPERTY

{attribute 'monitoring' := 'call'}
{attribute 'OPC.UA.DA.Property' := '1'}
{attribute 'OPC.UA.DA.Access' := '1'}
PROPERTY Error : BOOL
GET
Error := _Error;
END_GET
END_PROPERTY

METHOD Execute
_Busy := FALSE;
_Done := TRUE;
_Error := FALSE;
END_METHOD

{attribute 'monitoring' := 'call'}
{attribute 'OPC.UA.DA.Property' := '1'}
{attribute 'OPC.UA.DA.Access' := '1'}
PROPERTY ABSTRACT FromState : STRING
GET
END_GET
END_PROPERTY

METHOD Initialize
VAR_INPUT
	stateMachine : REFERENCE TO FiniteStateMachine;
END_VAR
IF NOT __ISVALIDREF(_StateMachine) THEN
	//exceptionFactory.ThrowException(__POSITION(), "programStateMachine is NULL");
END_IF

_StateMachine REF= stateMachine;
END_METHOD

{attribute 'monitoring' := 'call'}
{attribute 'OPC.UA.DA.Property' := '1'}
{attribute 'OPC.UA.DA.Access' := '1'}
PROPERTY Initialized : BOOL
GET
Initialized := __ISVALIDREF(_StateMachine);
END_GET
END_PROPERTY

{attribute 'monitoring' := 'call'}
PROPERTY LastException : REFERENCE TO Exception
GET
LastException REF= _LastException;
END_GET
END_PROPERTY

{attribute 'monitoring' := 'call'}
{attribute 'OPC.UA.DA.Property' := '1'}
{attribute 'OPC.UA.DA.Access' := '1'}
PROPERTY ABSTRACT Name : STRING
GET
END_GET
END_PROPERTY

METHOD Start
_Busy := FALSE;
_Done := TRUE;
_Error := FALSE;
END_METHOD

{attribute 'monitoring' := 'call'}
{attribute 'OPC.UA.DA.Property' := '1'}
{attribute 'OPC.UA.DA.Access' := '1'}
PROPERTY ABSTRACT ToState : STRING
GET
END_GET
END_PROPERTY

END_FUNCTION_BLOCK

// ---- StateMachine/Program/ProgramStateMachine.TcPOU
FUNCTION_BLOCK ABSTRACT ProgramStateMachine EXTENDS FiniteStateMachine
VAR
	{attribute 'OPC.UA.DA' := '0'}
	_HaltedState : REFERENCE TO HaltedProgramState;
	{attribute 'OPC.UA.DA' := '0'}
	_ReadyState : REFERENCE TO ReadyProgramState;
	{attribute 'OPC.UA.DA' := '0'}
	_RunningState : REFERENCE TO RunningProgramState;
	{attribute 'OPC.UA.DA' := '0'}
	_SuspendedState : REFERENCE TO SuspendedProgramState;
	
	{attribute 'OPC.UA.DA' := '0'}
	_HaltedToReady : REFERENCE TO HaltedToReadyProgramTransition;
	{attribute 'OPC.UA.DA' := '0'}
	_ReadyToRunning : REFERENCE TO ReadyToRunningProgramTransition;
	{attribute 'OPC.UA.DA' := '0'}
	_RunningToHalted : REFERENCE TO RunningToHaltedProgramTransition;
	{attribute 'OPC.UA.DA' := '0'}
	_RunningToReady : REFERENCE TO RunningToReadyProgramTransition;
	{attribute 'OPC.UA.DA' := '0'}
	_RunningToSuspended : REFERENCE TO RunningToSuspendedProgramTransition;
	{attribute 'OPC.UA.DA' := '0'}
	_SuspendedToRunning : REFERENCE TO SuspendedToRunningProgramTransition;
	{attribute 'OPC.UA.DA' := '0'}
	_SuspendedToHalted : REFERENCE TO SuspendedToHaltedProgramTransition;
	{attribute 'OPC.UA.DA' := '0'}
	_SuspendedToReady : REFERENCE TO SuspendedToReadyProgramTransition;
	{attribute 'OPC.UA.DA' := '0'}
	_ReadyToHalted : REFERENCE TO ReadyToHaltedProgramTransition;
END_VAR

{attribute 'monitoring' := 'call'}
{attribute 'OPC.UA.DA.Property' := '1'}
{attribute 'OPC.UA.DA.Access' := '1'}
PROPERTY AvailableStateCount : INT (0..(ProgramConstants.MaxStateCount - 1))
GET
AvailableStateCount := 4;
END_GET
END_PROPERTY

{attribute 'monitoring' := 'call'}
{attribute 'OPC.UA.DA.Property' := '1'}
{attribute 'OPC.UA.DA.Access' := '1'}
PROPERTY AvailableTransitionCount : INT (0..(ProgramConstants.MaxTransitionCount - 1))
GET
AvailableTransitionCount := 9;
END_GET
END_PROPERTY

METHOD PROTECTED ABSTRACT GetStateAndTransitionInstances
VAR_OUTPUT
	haltedState : POINTER TO HaltedProgramState;
	readyState : POINTER TO ReadyProgramState;
	runningState : POINTER TO RunningProgramState;
	suspendedState : POINTER TO SuspendedProgramState;
	
	haltedToReady : POINTER TO HaltedToReadyProgramTransition;
	readyToRunning : POINTER TO ReadyToRunningProgramTransition;
	runningToHalted : POINTER TO RunningToHaltedProgramTransition;
	runningToReady : POINTER TO RunningToReadyProgramTransition;
	runningToSuspended : POINTER TO RunningToSuspendedProgramTransition;
	suspendedToRunning : POINTER TO SuspendedToRunningProgramTransition;
	suspendedToHalted : POINTER TO SuspendedToHaltedProgramTransition;
	suspendedToReady : POINTER TO SuspendedToReadyProgramTransition;
	readyToHalted : POINTER TO ReadyToHaltedProgramTransition;	
END_VAR
END_METHOD

{attribute 'TcRpcEnable':='1'}
METHOD FINAL Halt : BOOL
VAR_OUTPUT
	errorMessage : ERROR_MESSAGE;
END_VAR
__TRY
	FindTransitionByCause(__POUNAME());
	RequestedCause := __POUNAME();
	Halt := TRUE;
__CATCH
	errorMessage := ExceptionHelper.LastException.ToString(FALSE);
	ExceptionHelper.Cleanup();
__ENDTRY
END_METHOD

METHOD PROTECTED InternalInitialize 
VAR_OUTPUT
	states : ARRAY [0..ProgramConstants.MaxStateCount - 1] OF POINTER TO ProgramState;
	transitions : ARRAY [0..ProgramConstants.MaxTransitionCount - 1] OF POINTER TO ProgramTransition;
	defaultState : POINTER TO ProgramState;
END_VAR
VAR
	haltedState : POINTER TO HaltedProgramState;
	readyState : POINTER TO ReadyProgramState;
	runningState : POINTER TO RunningProgramState;
	suspendedState : POINTER TO SuspendedProgramState;
	
	haltedToReady : POINTER TO HaltedToReadyProgramTransition;
	readyToRunning : POINTER TO ReadyToRunningProgramTransition;
	runningToHalted : POINTER TO RunningToHaltedProgramTransition;
	runningToReady : POINTER TO RunningToReadyProgramTransition;
	runningToSuspended : POINTER TO RunningToSuspendedProgramTransition;
	suspendedToRunning : POINTER TO SuspendedToRunningProgramTransition;
	suspendedToHalted : POINTER TO SuspendedToHaltedProgramTransition;
	suspendedToReady : POINTER TO SuspendedToReadyProgramTransition;
	readyToHalted : POINTER TO ReadyToHaltedProgramTransition;	
END_VAR
GetStateAndTransitionInstances(	
	haltedState => haltedState, 
	readyState => readyState, 
	runningState => runningState, 
	suspendedState => suspendedState,
	
	haltedToReady => haltedToReady,
	readyToRunning => readyToRunning,
	runningToHalted => runningToHalted,
	runningToReady => runningToReady,
	runningToSuspended => runningToSuspended,
	suspendedToRunning => suspendedToRunning,
	suspendedToHalted => suspendedToHalted,
	suspendedToReady => suspendedToReady,
	readyToHalted => readyToHalted
);	

_HaltedState REF= haltedState^;
_ReadyState REF= readyState^;
_RunningState REF= runningState^;
_SuspendedState REF= suspendedState^;

_HaltedToReady REF= haltedToReady^;
_ReadyToRunning REF= readyToRunning^;
_RunningToHalted REF= runningToHalted^;
_RunningToReady REF= runningToReady^;
_RunningToSuspended REF= runningToSuspended^;
_SuspendedToRunning REF= suspendedToRunning^;
_SuspendedToHalted REF= suspendedToHalted^;
_SuspendedToReady REF= suspendedToReady^;
_ReadyToHalted REF= readyToHalted^;

states[0] := haltedState;
states[1] := readyState;
states[2] := runningState;
states[3] := suspendedState;

transitions[0] := haltedToReady;
transitions[1] := readyToRunning;
transitions[2] := runningToHalted;
transitions[3] := runningToReady;
transitions[4] := runningToSuspended;
transitions[5] := suspendedToRunning;
transitions[6] := suspendedToHalted;
transitions[7] := suspendedToReady;
transitions[8] := readyToHalted;

defaultState := readyState;
END_METHOD

{attribute 'TcRpcEnable':='1'}
METHOD FINAL Reset : BOOL
VAR_OUTPUT
	errorMessage : ERROR_MESSAGE;
END_VAR
__TRY
	FindTransitionByCause(__POUNAME());
	RequestedCause := __POUNAME();
	Reset := TRUE;
__CATCH
	errorMessage := ExceptionHelper.LastException.ToString(FALSE);
	ExceptionHelper.Cleanup();
__ENDTRY
END_METHOD

{attribute 'TcRpcEnable':='1'}
METHOD FINAL Resume : BOOL
VAR_OUTPUT
	errorMessage : ERROR_MESSAGE;
END_VAR
__TRY
	FindTransitionByCause(__POUNAME());
	RequestedCause := __POUNAME();
	Resume := TRUE;	
__CATCH
	errorMessage := ExceptionHelper.LastException.ToString(FALSE);
	ExceptionHelper.Cleanup();
__ENDTRY
END_METHOD

{attribute 'TcRpcEnable':='1'}
METHOD FINAL Start: BOOL
VAR_OUTPUT
	errorMessage : ERROR_MESSAGE;
END_VAR
__TRY
	FindTransitionByCause(__POUNAME());
	RequestedCause := __POUNAME();
	Start := TRUE;
__CATCH
	errorMessage := ExceptionHelper.LastException.ToString(FALSE);
	ExceptionHelper.Cleanup();
__ENDTRY
END_METHOD

{attribute 'TcRpcEnable':='1'}
METHOD FINAL Suspend : BOOL
VAR_OUTPUT
	errorMessage : ERROR_MESSAGE;
END_VAR
__TRY
	FindTransitionByCause(__POUNAME());
	RequestedCause := __POUNAME();
	Suspend := TRUE;
__CATCH
	errorMessage := ExceptionHelper.LastException.ToString(FALSE);
	ExceptionHelper.Cleanup();
__ENDTRY
END_METHOD

END_FUNCTION_BLOCK

// ---- StateMachine/Program/States/HaltedProgramState.TcPOU
FUNCTION_BLOCK ABSTRACT HaltedProgramState EXTENDS ProgramState

{attribute 'monitoring' := 'call'}
{attribute 'OPC.UA.DA.Property' := '1'}
{attribute 'OPC.UA.DA.Access' := '1'}
PROPERTY FINAL Name : STRING
GET
Name := 'Halted';
END_GET
END_PROPERTY

END_FUNCTION_BLOCK

// ---- StateMachine/Program/States/ReadyProgramState.TcPOU
FUNCTION_BLOCK ABSTRACT ReadyProgramState EXTENDS ProgramState

{attribute 'monitoring' := 'call'}
{attribute 'OPC.UA.DA.Property' := '1'}
{attribute 'OPC.UA.DA.Access' := '1'}
PROPERTY FINAL Name : STRING
GET
Name := 'Ready';
END_GET
END_PROPERTY

END_FUNCTION_BLOCK

// ---- StateMachine/Program/States/RunningProgramState.TcPOU
FUNCTION_BLOCK ABSTRACT RunningProgramState EXTENDS ProgramState

{attribute 'monitoring' := 'call'}
{attribute 'OPC.UA.DA.Property' := '1'}
{attribute 'OPC.UA.DA.Access' := '1'}
PROPERTY FINAL Name : STRING
GET
Name := 'Running';
END_GET
END_PROPERTY

END_FUNCTION_BLOCK

// ---- StateMachine/Program/States/SuspendedProgramState.TcPOU
FUNCTION_BLOCK ABSTRACT SuspendedProgramState EXTENDS ProgramState

{attribute 'monitoring' := 'call'}
{attribute 'OPC.UA.DA.Property' := '1'}
{attribute 'OPC.UA.DA.Access' := '1'}
PROPERTY FINAL Name : STRING
GET
Name := 'Suspended';
END_GET
END_PROPERTY

END_FUNCTION_BLOCK

// ---- StateMachine/Program/Transitions/HaltedToReadyProgramTransition.TcPOU
FUNCTION_BLOCK ABSTRACT HaltedToReadyProgramTransition EXTENDS ProgramTransition

{attribute 'monitoring' := 'call'}
{attribute 'OPC.UA.DA.Property' := '1'}
{attribute 'OPC.UA.DA.Access' := '1'}
PROPERTY FINAL Cause : STRING
GET
Cause := 'Reset';
END_GET
END_PROPERTY

{attribute 'monitoring' := 'call'}
{attribute 'OPC.UA.DA.Property' := '1'}
{attribute 'OPC.UA.DA.Access' := '1'}
PROPERTY FINAL FromState : STRING
GET
FromState := 'Halted';
END_GET
END_PROPERTY

{attribute 'monitoring' := 'call'}
{attribute 'OPC.UA.DA.Property' := '1'}
{attribute 'OPC.UA.DA.Access' := '1'}
PROPERTY FINAL Name : STRING
GET
Name := 'HaltedToReady';
END_GET
END_PROPERTY

{attribute 'monitoring' := 'call'}
{attribute 'OPC.UA.DA.Property' := '1'}
{attribute 'OPC.UA.DA.Access' := '1'}
PROPERTY FINAL ToState : STRING
GET
ToState := 'Ready';
END_GET
END_PROPERTY

END_FUNCTION_BLOCK

// ---- StateMachine/Program/Transitions/ReadyToRunningProgramTransition.TcPOU
FUNCTION_BLOCK ABSTRACT ReadyToRunningProgramTransition EXTENDS ProgramTransition

{attribute 'monitoring' := 'call'}
{attribute 'OPC.UA.DA.Property' := '1'}
{attribute 'OPC.UA.DA.Access' := '1'}
PROPERTY FINAL Cause : STRING
GET
Cause := 'Start';
END_GET
END_PROPERTY

{attribute 'monitoring' := 'call'}
{attribute 'OPC.UA.DA.Property' := '1'}
{attribute 'OPC.UA.DA.Access' := '1'}
PROPERTY FINAL FromState : STRING
GET
FromState := 'Ready';
END_GET
END_PROPERTY

{attribute 'monitoring' := 'call'}
{attribute 'OPC.UA.DA.Property' := '1'}
{attribute 'OPC.UA.DA.Access' := '1'}
PROPERTY FINAL Name : STRING
GET
Name := 'ReadyToRunning';
END_GET
END_PROPERTY

{attribute 'monitoring' := 'call'}
{attribute 'OPC.UA.DA.Property' := '1'}
{attribute 'OPC.UA.DA.Access' := '1'}
PROPERTY FINAL ToState : STRING
GET
ToState := 'Running';
END_GET
END_PROPERTY

END_FUNCTION_BLOCK

// ---- StateMachine/Program/Transitions/RunningToHaltedProgramTransition.TcPOU
FUNCTION_BLOCK ABSTRACT RunningToHaltedProgramTransition EXTENDS ProgramTransition

{attribute 'monitoring' := 'call'}
{attribute 'OPC.UA.DA.Property' := '1'}
{attribute 'OPC.UA.DA.Access' := '1'}
PROPERTY FINAL Cause : STRING
GET
Cause := 'Halt';
END_GET
END_PROPERTY

{attribute 'monitoring' := 'call'}
{attribute 'OPC.UA.DA.Property' := '1'}
{attribute 'OPC.UA.DA.Access' := '1'}
PROPERTY FINAL FromState : STRING
GET
FromState := 'Running';
END_GET
END_PROPERTY

{attribute 'monitoring' := 'call'}
{attribute 'OPC.UA.DA.Property' := '1'}
{attribute 'OPC.UA.DA.Access' := '1'}
PROPERTY FINAL Name : STRING
GET
Name := 'RunningToHalted';
END_GET
END_PROPERTY

{attribute 'monitoring' := 'call'}
{attribute 'OPC.UA.DA.Property' := '1'}
{attribute 'OPC.UA.DA.Access' := '1'}
PROPERTY FINAL ToState : STRING
GET
ToState := 'Halted';
END_GET
END_PROPERTY

END_FUNCTION_BLOCK

// ---- StateMachine/Program/Transitions/RunningToReadyProgramTransition.TcPOU
FUNCTION_BLOCK ABSTRACT RunningToReadyProgramTransition EXTENDS ProgramTransition

{attribute 'monitoring' := 'call'}
{attribute 'OPC.UA.DA.Property' := '1'}
{attribute 'OPC.UA.DA.Access' := '1'}
PROPERTY FINAL Cause : STRING
GET
Cause := '';
END_GET
END_PROPERTY

{attribute 'monitoring' := 'call'}
{attribute 'OPC.UA.DA.Property' := '1'}
{attribute 'OPC.UA.DA.Access' := '1'}
PROPERTY FINAL FromState : STRING
GET
FromState := 'Running';
END_GET
END_PROPERTY

{attribute 'monitoring' := 'call'}
{attribute 'OPC.UA.DA.Property' := '1'}
{attribute 'OPC.UA.DA.Access' := '1'}
PROPERTY FINAL Name : STRING
GET
Name := 'RunningToReady';
END_GET
END_PROPERTY

{attribute 'monitoring' := 'call'}
{attribute 'OPC.UA.DA.Property' := '1'}
{attribute 'OPC.UA.DA.Access' := '1'}
PROPERTY FINAL ToState : STRING
GET
ToState := 'Ready';
END_GET
END_PROPERTY

END_FUNCTION_BLOCK

// ---- StateMachine/Program/Transitions/RunningToSuspendedProgramTransition.TcPOU
FUNCTION_BLOCK ABSTRACT RunningToSuspendedProgramTransition EXTENDS ProgramTransition

{attribute 'monitoring' := 'call'}
{attribute 'OPC.UA.DA.Property' := '1'}
{attribute 'OPC.UA.DA.Access' := '1'}
PROPERTY FINAL Cause : STRING
GET
Cause := 'Suspend';
END_GET
END_PROPERTY

{attribute 'monitoring' := 'call'}
{attribute 'OPC.UA.DA.Property' := '1'}
{attribute 'OPC.UA.DA.Access' := '1'}
PROPERTY FINAL FromState : STRING
GET
FromState := 'Running';
END_GET
END_PROPERTY

{attribute 'monitoring' := 'call'}
{attribute 'OPC.UA.DA.Property' := '1'}
{attribute 'OPC.UA.DA.Access' := '1'}
PROPERTY FINAL Name : STRING
GET
Name := 'RunningToSuspended';
END_GET
END_PROPERTY

{attribute 'monitoring' := 'call'}
{attribute 'OPC.UA.DA.Property' := '1'}
{attribute 'OPC.UA.DA.Access' := '1'}
PROPERTY FINAL ToState : STRING
GET
ToState := 'Suspended';
END_GET
END_PROPERTY

END_FUNCTION_BLOCK

// ---- StateMachine/Program/Transitions/SuspendedToRunningProgramTransition.TcPOU
FUNCTION_BLOCK ABSTRACT SuspendedToRunningProgramTransition EXTENDS ProgramTransition

{attribute 'monitoring' := 'call'}
{attribute 'OPC.UA.DA.Property' := '1'}
{attribute 'OPC.UA.DA.Access' := '1'}
PROPERTY FINAL Cause : STRING
GET
Cause := 'Resume';
END_GET
END_PROPERTY

{attribute 'monitoring' := 'call'}
{attribute 'OPC.UA.DA.Property' := '1'}
{attribute 'OPC.UA.DA.Access' := '1'}
PROPERTY FINAL FromState : STRING
GET
FromState := 'Suspended';
END_GET
END_PROPERTY

{attribute 'monitoring' := 'call'}
{attribute 'OPC.UA.DA.Property' := '1'}
{attribute 'OPC.UA.DA.Access' := '1'}
PROPERTY FINAL Name : STRING
GET
Name := 'SuspendedToRunning';
END_GET
END_PROPERTY

{attribute 'monitoring' := 'call'}
{attribute 'OPC.UA.DA.Property' := '1'}
{attribute 'OPC.UA.DA.Access' := '1'}
PROPERTY FINAL ToState : STRING
GET
ToState := 'Running';
END_GET
END_PROPERTY

END_FUNCTION_BLOCK

// ---- StateMachine/Program/Transitions/SuspendedToHaltedProgramTransition.TcPOU
FUNCTION_BLOCK ABSTRACT SuspendedToHaltedProgramTransition EXTENDS ProgramTransition

{attribute 'monitoring' := 'call'}
{attribute 'OPC.UA.DA.Property' := '1'}
{attribute 'OPC.UA.DA.Access' := '1'}
PROPERTY FINAL Cause : STRING
GET
Cause := 'Halt';
END_GET
END_PROPERTY

{attribute 'monitoring' := 'call'}
{attribute 'OPC.UA.DA.Property' := '1'}
{attribute 'OPC.UA.DA.Access' := '1'}
PROPERTY FINAL FromState : STRING
GET
FromState := 'Suspended';
END_GET
END_PROPERTY

{attribute 'monitoring' := 'call'}
{attribute 'OPC.UA.DA.Property' := '1'}
{attribute 'OPC.UA.DA.Access' := '1'}
PROPERTY FINAL Name : STRING
GET
Name := 'SuspendedToHalted';
END_GET
END_PROPERTY

{attribute 'monitoring' := 'call'}
{attribute 'OPC.UA.DA.Property' := '1'}
{attribute 'OPC.UA.DA.Access' := '1'}
PROPERTY FINAL ToState : STRING
GET
ToState := 'Halted';
END_GET
END_PROPERTY

END_FUNCTION_BLOCK

// ---- StateMachine/Program/Transitions/SuspendedToReadyProgramTransition.TcPOU
FUNCTION_BLOCK ABSTRACT SuspendedToReadyProgramTransition EXTENDS ProgramTransition

{attribute 'monitoring' := 'call'}
{attribute 'OPC.UA.DA.Property' := '1'}
{attribute 'OPC.UA.DA.Access' := '1'}
PROPERTY FINAL Cause : STRING
GET
Cause := 'Reset';
END_GET
END_PROPERTY

{attribute 'monitoring' := 'call'}
{attribute 'OPC.UA.DA.Property' := '1'}
{attribute 'OPC.UA.DA.Access' := '1'}
PROPERTY FINAL FromState : STRING
GET
FromState := 'Suspended';
END_GET
END_PROPERTY

{attribute 'monitoring' := 'call'}
{attribute 'OPC.UA.DA.Property' := '1'}
{attribute 'OPC.UA.DA.Access' := '1'}
PROPERTY FINAL Name : STRING
GET
Name := 'SuspendedToReady';
END_GET
END_PROPERTY

{attribute 'monitoring' := 'call'}
{attribute 'OPC.UA.DA.Property' := '1'}
{attribute 'OPC.UA.DA.Access' := '1'}
PROPERTY FINAL ToState : STRING
GET
ToState := 'Ready';
END_GET
END_PROPERTY

END_FUNCTION_BLOCK

// ---- StateMachine/Program/Transitions/ReadyToHaltedProgramTransition.TcPOU
FUNCTION_BLOCK ABSTRACT ReadyToHaltedProgramTransition EXTENDS ProgramTransition

{attribute 'monitoring' := 'call'}
{attribute 'OPC.UA.DA.Property' := '1'}
{attribute 'OPC.UA.DA.Access' := '1'}
PROPERTY FINAL Cause : STRING
GET
Cause := '';
END_GET
END_PROPERTY

{attribute 'monitoring' := 'call'}
{attribute 'OPC.UA.DA.Property' := '1'}
{attribute 'OPC.UA.DA.Access' := '1'}
PROPERTY FINAL FromState : STRING
GET
FromState := '';
END_GET
END_PROPERTY

{attribute 'monitoring' := 'call'}
{attribute 'OPC.UA.DA.Property' := '1'}
{attribute 'OPC.UA.DA.Access' := '1'}
PROPERTY FINAL Name : STRING
GET
Name := 'ReadyToHalted';
END_GET
END_PROPERTY

{attribute 'monitoring' := 'call'}
{attribute 'OPC.UA.DA.Property' := '1'}
{attribute 'OPC.UA.DA.Access' := '1'}
PROPERTY FINAL ToState : STRING
GET
ToState := 'Halted';
END_GET
END_PROPERTY

END_FUNCTION_BLOCK

// ---- StateMachine/UnifiedProgram/States/HaltedUnifiedProgramState.TcPOU
FUNCTION_BLOCK HaltedUnifiedProgramState EXTENDS HaltedProgramState
VAR
	{attribute 'OPC.UA.DA' := '0'}
	_ClassName : STRING := __POUNAME();
END_VAR

{attribute 'monitoring' := 'call'}
PROPERTY ClassName : STRING
GET
ClassName := _ClassName;
END_GET
END_PROPERTY

END_FUNCTION_BLOCK

// ---- StateMachine/UnifiedProgram/States/ReadyUnifiedProgramState.TcPOU
FUNCTION_BLOCK ReadyUnifiedProgramState EXTENDS ReadyProgramState
VAR
	{attribute 'OPC.UA.DA' := '0'}
	_ClassName : STRING := __POUNAME();
END_VAR

{attribute 'monitoring' := 'call'}
PROPERTY ClassName : STRING
GET
ClassName := _ClassName;
END_GET
END_PROPERTY

END_FUNCTION_BLOCK

// ---- StateMachine/UnifiedProgram/States/RunningUnifiedProgramState.TcPOU
FUNCTION_BLOCK RunningUnifiedProgramState EXTENDS RunningProgramState
VAR
	{attribute 'OPC.UA.DA' := '0'}
	_ClassName : STRING := __POUNAME();
END_VAR

{attribute 'monitoring' := 'call'}
PROPERTY ClassName : STRING
GET
ClassName := _ClassName;
END_GET
END_PROPERTY

END_FUNCTION_BLOCK

// ---- StateMachine/UnifiedProgram/States/SuspendedUnifiedProgramState.TcPOU
FUNCTION_BLOCK SuspendedUnifiedProgramState EXTENDS SuspendedProgramState
VAR
	{attribute 'OPC.UA.DA' := '0'}
	_ClassName : STRING := __POUNAME();
END_VAR

{attribute 'monitoring' := 'call'}
PROPERTY ClassName : STRING
GET
ClassName := _ClassName;
END_GET
END_PROPERTY

END_FUNCTION_BLOCK

// ---- StateMachine/UnifiedProgram/StepModels/UnifiedProgramExecutedStep.TcPOU
FUNCTION_BLOCK UnifiedProgramExecutedStep EXTENDS ToolkitObject
VAR_OUTPUT
	StepIndex : INT;
	
	Suspend : BOOL;
	Complete : BOOL;
	
	Actions : ARRAY [0..UnifiedProgramConstants.MaxStepActionsCount - 1] OF POINTER TO UnifiedProgramExecutedStepAction;
	ActionCount : INT;
	
	Transitions : ARRAY [0..UnifiedProgramConstants.MaxStepTransitionsCount - 1] OF POINTER TO UnifiedProgramExecutedStepTransition;
	TransitionCount : INT;
END_VAR
VAR
	{attribute 'OPC.UA.DA' := '0'}
	_ClassName : STRING := __POUNAME();
END_VAR

{attribute 'monitoring' := 'call'}
PROPERTY ClassName : STRING
GET
ClassName := _ClassName;
END_GET
END_PROPERTY

METHOD Clear
VAR
	i : INT;
END_VAR
Suspend := FALSE;
Complete := FALSE;

FOR i := 0 TO UnifiedProgramConstants.MaxStepActionsCount - 1 DO
	IF Actions[i] <> 0 THEN
		__DELETE(Actions[i]);		
	END_IF
END_FOR

ActionCount := 0;

FOR i := 0 TO UnifiedProgramConstants.MaxStepTransitionsCount - 1 DO
	IF Transitions[i] <> 0 THEN
		__DELETE(Actions[i]);		
	END_IF	
END_FOR

TransitionCount := 0;
END_METHOD

METHOD Decode : BOOL
VAR_INPUT
	stepIndex : INT; 
	step : REFERENCE TO UNIFIED_PROGRAM_STEP;
END_VAR
VAR
	i : INT;
END_VAR
StepIndex := stepIndex;	
Suspend := step.Suspend;
Complete := step.Complete;

FOR i := 0 TO UnifiedProgramConstants.MaxStepActionsCount - 1 DO
	IF step.Actions[i].Name <> '' THEN
		Actions[i] := UnifiedProgramExecutedStepHelper.CreateActionInstance(step.Actions[i].Name, exception => exception);
		
		IF Actions[i] = 0 THEN
			RETURN;
		END_IF
		
		IF NOT Actions[i]^.Decode(i, step.Actions[i], exception => exception) THEN
			RETURN;
		END_IF
	ELSE
		EXIT;
	END_IF
END_FOR

(*FOR i := 0 TO UnifiedProgramConstants.MaxStepTransitionsCount - 1 DO
		Transitions[i] := UnifiedProgramExecutedStepHelper.CreateActionInstance(step.Actions[i].Name, exception => exception);
		
		IF Actions[i] = 0 THEN
			RETURN;
		END_IF
		
		IF NOT Actions[i]^.Decode(i, step.Actions[i], exception => exception) THEN
			RETURN;
		END_IF
	ELSE
		EXIT;
	END_IF
END_FOR*)
END_METHOD

END_FUNCTION_BLOCK

// ---- StateMachine/UnifiedProgram/StepModels/UnifiedProgramExecutedStepAction.TcPOU
FUNCTION_BLOCK ABSTRACT UnifiedProgramExecutedStepAction EXTENDS ToolkitObject
VAR
	{attribute 'OPC.UA.DA' := '0'}
	_ClassName : STRING := __POUNAME();
END_VAR

METHOD ABSTRACT Decode : BOOL
VAR_INPUT
	actionIndex : INT; 
	stepAction : REFERENCE TO UNIFIED_PROGRAM_STEP_ACTION;
END_VAR
END_METHOD

END_FUNCTION_BLOCK

// ---- StateMachine/UnifiedProgram/StepModels/UnifiedProgramExecutedStepTransition.TcPOU
FUNCTION_BLOCK UnifiedProgramExecutedStepTransition EXTENDS ToolkitObject
VAR
	{attribute 'OPC.UA.DA' := '0'}
	_ClassName : STRING := __POUNAME();
END_VAR

{attribute 'monitoring' := 'call'}
PROPERTY ClassName : STRING
GET
ClassName := _ClassName;
END_GET
END_PROPERTY

METHOD Decode : BOOL
VAR_INPUT
	transitionIndex : INT; 
	stepTransition : REFERENCE TO UNIFIED_PROGRAM_STEP_TRANSITION;
END_VAR
END_METHOD

END_FUNCTION_BLOCK

// ---- StateMachine/UnifiedProgram/StepModels/UnifiedProgramExecutedStepHelper.TcPOU
PROGRAM UnifiedProgramExecutedStepHelper

METHOD CreateActionInstance : POINTER TO UnifiedProgramExecutedStepAction
VAR_INPUT
	actionName : STRING;
END_VAR
END_METHOD

METHOD CreateTransitionConditionInstance : POINTER TO UnifiedProgramExecutedStepTransitionCondition
VAR_INPUT
	conditionName : STRING;
END_VAR
END_METHOD

END_PROGRAM

// ---- StateMachine/UnifiedProgram/StepModels/UnifiedProgramExecutedStepTransitionCondition.TcPOU
FUNCTION_BLOCK ABSTRACT UnifiedProgramExecutedStepTransitionCondition EXTENDS ToolkitObject
VAR
	{attribute 'OPC.UA.DA' := '0'}
	_ClassName : STRING := __POUNAME();
END_VAR

METHOD ABSTRACT Decode : BOOL
VAR_INPUT
	transitionIndex : INT; 
	stepTransition : REFERENCE TO UNIFIED_PROGRAM_STEP_TRANSITION;
END_VAR
END_METHOD

END_FUNCTION_BLOCK

// ---- StateMachine/UnifiedProgram/Transitions/HaltedToReadyUnifiedProgramTransition.TcPOU
FUNCTION_BLOCK HaltedToReadyUnifiedProgramTransition EXTENDS HaltedToReadyProgramTransition
VAR
	{attribute 'OPC.UA.DA' := '0'}
	_ClassName : STRING := __POUNAME();
END_VAR

{attribute 'monitoring' := 'call'}
PROPERTY ClassName : STRING
GET
ClassName := _ClassName;
END_GET
END_PROPERTY

END_FUNCTION_BLOCK

// ---- StateMachine/UnifiedProgram/Transitions/ReadyToHaltedUnifiedProgramTransition.TcPOU
FUNCTION_BLOCK ReadyToHaltedUnifiedProgramTransition EXTENDS ReadyToHaltedProgramTransition
VAR
	{attribute 'OPC.UA.DA' := '0'}
	_ClassName : STRING := __POUNAME();
END_VAR

{attribute 'monitoring' := 'call'}
PROPERTY ClassName : STRING
GET
ClassName := _ClassName;
END_GET
END_PROPERTY

END_FUNCTION_BLOCK

// ---- StateMachine/UnifiedProgram/Transitions/ReadyToRunningUnifiedProgramTransition.TcPOU
FUNCTION_BLOCK ReadyToRunningUnifiedProgramTransition EXTENDS ReadyToRunningProgramTransition
VAR
	{attribute 'OPC.UA.DA' := '0'}
	_ClassName : STRING := __POUNAME();
END_VAR

{attribute 'monitoring' := 'call'}
PROPERTY ClassName : STRING
GET
ClassName := _ClassName;
END_GET
END_PROPERTY

METHOD Start
VAR
	i : INT;
	executedSteps : ARRAY [0..UnifiedProgramConstants.MaxStepCount - 1] OF UNIFIED_PROGRAM_EXECUTED_STEP;
	executedStepCount : INT;
END_VAR
UnifiedProgramStateMachine^.LastException.Clear();
UnifiedProgramStateMachine^.StepExecutor.Reset();

FOR i := 0 TO UnifiedProgramConstants.MaxStepCount - 1 DO
	executedSteps[i].StepIndex := i;
	ExecutedSteps[i].Step REF= UnifiedProgramStateMachine^.Configuration.Steps[i];
	
	executedStepCount := executedStepCount + 1;
	
	IF UnifiedProgramStateMachine^.Configuration.Steps[i].Complete THEN
		EXIT;
	END_IF
END_FOR

_Busy := FALSE;
_Done := TRUE;
_Error := FALSE;
END_METHOD

PROPERTY UnifiedProgramStateMachine : POINTER TO UnifiedProgramStateMachine
GET
UnifiedProgramStateMachine := ADR(_StateMachine);
END_GET
END_PROPERTY

END_FUNCTION_BLOCK

// ---- StateMachine/UnifiedProgram/UnifiedProgramStateMachine.TcPOU
{attribute 'no_explicit_call' := 'do not call this function block directly'} 
FUNCTION_BLOCK UnifiedProgramStateMachine EXTENDS ProgramStateMachine
VAR_OUTPUT
	{attribute 'OPC.UA.DA.Access' := '1'}
	Configuration : UNIFIED_PROGRAM_CONFIGURATION;
	
	{attribute 'OPC.UA.DA.Access' := '1'}
	HaltedState : HaltedUnifiedProgramState;
	{attribute 'OPC.UA.DA.Access' := '1'}
	ReadyState : ReadyUnifiedProgramState;
	{attribute 'OPC.UA.DA.Access' := '1'}
	RunningState : RunningUnifiedProgramState;
	{attribute 'OPC.UA.DA.Access' := '1'}
	SuspendedState : SuspendedUnifiedProgramState;
	
	{attribute 'OPC.UA.DA.Access' := '1'}
	HaltedToReady : HaltedToReadyUnifiedProgramTransition;
	{attribute 'OPC.UA.DA.Access' := '1'}
	ReadyToRunning : ReadyToRunningUnifiedProgramTransition;
	{attribute 'OPC.UA.DA.Access' := '1'}
	RunningToHalted : RunningToHaltedUnifiedProgramTransition;
	{attribute 'OPC.UA.DA.Access' := '1'}
	RunningToReady : RunningToReadyUnifiedProgramTransition;
	{attribute 'OPC.UA.DA.Access' := '1'}
	RunningToSuspended : RunningToSuspendedUnifiedProgramTransition;
	{attribute 'OPC.UA.DA.Access' := '1'}
	SuspendedToRunning : SuspendedToRunningUnifiedProgramTransition;
	{attribute 'OPC.UA.DA.Access' := '1'}
	SuspendedToHalted : SuspendedToHaltedUnifiedProgramTransition;
	{attribute 'OPC.UA.DA.Access' := '1'}
	SuspendedToReady : SuspendedToReadyUnifiedProgramTransition;
	{attribute 'OPC.UA.DA.Access' := '1'}
	ReadyToHalted : ReadyToHaltedUnifiedProgramTransition;
	
	{attribute 'OPC.UA.DA' := '0'}
	StepExecutor : UnifiedProgramStepExecutor(THIS^);
END_VAR
VAR
	{attribute 'OPC.UA.DA' := '0'}
	_ClassName : STRING := __POUNAME();
END_VAR

{attribute 'monitoring' := 'call'}
PROPERTY ClassName : STRING
GET
ClassName := _ClassName;
END_GET
END_PROPERTY

METHOD FB_init : BOOL
VAR_INPUT
	bInitRetains : BOOL; // if TRUE, the retain variables are initialized (warm start / cold start)
	bInCopyCode : BOOL;  // if TRUE, the instance afterwards gets moved into the copy code (online change)
END_VAR
JsonHelper.SetFormatOptions(10, EJsonPrettyFormatOptions.eFormatSingleLineArray, 9, 1);
END_METHOD

{attribute 'TcRpcEnable':='1'}
METHOD GetConfiguration : JSON_DOCUMENT
JsonHelper.CreateJsonFromStructure(ADR(Configuration), SIZEOF(Configuration), GetConfiguration);
END_METHOD

METHOD PROTECTED GetStateAndTransitionInstances
VAR_OUTPUT
	haltedState : POINTER TO HaltedProgramState;
	readyState : POINTER TO ReadyProgramState;
	runningState : POINTER TO RunningProgramState;
	suspendedState : POINTER TO SuspendedProgramState;
	
	haltedToReady : POINTER TO HaltedToReadyProgramTransition;
	readyToRunning : POINTER TO ReadyToRunningProgramTransition;
	runningToHalted : POINTER TO RunningToHaltedProgramTransition;
	runningToReady : POINTER TO RunningToReadyProgramTransition;
	runningToSuspended : POINTER TO RunningToSuspendedProgramTransition;
	suspendedToRunning : POINTER TO SuspendedToRunningProgramTransition;
	suspendedToHalted : POINTER TO SuspendedToHaltedProgramTransition;
	suspendedToReady : POINTER TO SuspendedToReadyProgramTransition;
	readyToHalted : POINTER TO ReadyToHaltedProgramTransition;	
END_VAR
haltedState := ADR(THIS^.HaltedState);
readyState := ADR(THIS^.ReadyState);
runningState := ADR(THIS^.RunningState);
suspendedState := ADR(THIS^.SuspendedState);

haltedToReady := ADR(THIS^.HaltedToReady);
readyToRunning := ADR(THIS^.ReadyToRunning);
runningToHalted := ADR(THIS^.RunningToHalted);
runningToReady := ADR(THIS^.RunningToReady);
runningToSuspended := ADR(THIS^.RunningToSuspended);
suspendedToRunning := ADR(THIS^.SuspendedToRunning);
suspendedToHalted := ADR(THIS^.SuspendedToHalted);
suspendedToReady := ADR(THIS^.SuspendedToReady);
readyToHalted := ADR(THIS^.ReadyToHalted);
END_METHOD

METHOD PROTECTED InternalInitialize 
VAR_OUTPUT
	states : ARRAY [0..ProgramConstants.MaxStateCount - 1] OF POINTER TO ProgramState;
	transitions : ARRAY [0..ProgramConstants.MaxTransitionCount - 1] OF POINTER TO ProgramTransition;
	defaultState : POINTER TO ProgramState;
END_VAR
VAR
	haltedState : POINTER TO HaltedProgramState;
	readyState : POINTER TO ReadyProgramState;
	runningState : POINTER TO RunningProgramState;
	suspendedState : POINTER TO SuspendedProgramState;
	
	haltedToReady : POINTER TO HaltedToReadyProgramTransition;
	readyToRunning : POINTER TO ReadyToRunningProgramTransition;
	runningToHalted : POINTER TO RunningToHaltedProgramTransition;
	runningToReady : POINTER TO RunningToReadyProgramTransition;
	runningToSuspended : POINTER TO RunningToSuspendedProgramTransition;
	suspendedToRunning : POINTER TO SuspendedToRunningProgramTransition;
	suspendedToHalted : POINTER TO SuspendedToHaltedProgramTransition;
	suspendedToReady : POINTER TO SuspendedToReadyProgramTransition;
	readyToHalted : POINTER TO ReadyToHaltedProgramTransition;	
END_VAR
END_METHOD

{attribute 'TcRpcEnable':='1'}
METHOD SetConfiguration
VAR_INPUT
	json : JSON_DOCUMENT;
END_VAR
JsonHelper.SetStructureFromJson(json, ADR(Configuration), SIZEOF(Configuration));
END_METHOD

END_FUNCTION_BLOCK

// ---- StateMachine/UnifiedProgram/Transitions/RunningToHaltedUnifiedProgramTransition.TcPOU
FUNCTION_BLOCK RunningToHaltedUnifiedProgramTransition EXTENDS RunningToHaltedProgramTransition
VAR
	{attribute 'OPC.UA.DA' := '0'}
	_ClassName : STRING := __POUNAME();
END_VAR

{attribute 'monitoring' := 'call'}
PROPERTY ClassName : STRING
GET
ClassName := _ClassName;
END_GET
END_PROPERTY

END_FUNCTION_BLOCK

// ---- StateMachine/UnifiedProgram/Transitions/RunningToReadyUnifiedProgramTransition.TcPOU
FUNCTION_BLOCK RunningToReadyUnifiedProgramTransition EXTENDS RunningToReadyProgramTransition
VAR
	{attribute 'OPC.UA.DA' := '0'}
	_ClassName : STRING := __POUNAME();
END_VAR

{attribute 'monitoring' := 'call'}
PROPERTY ClassName : STRING
GET
ClassName := _ClassName;
END_GET
END_PROPERTY

END_FUNCTION_BLOCK

// ---- StateMachine/UnifiedProgram/Transitions/RunningToSuspendedUnifiedProgramTransition.TcPOU
FUNCTION_BLOCK RunningToSuspendedUnifiedProgramTransition EXTENDS RunningToSuspendedProgramTransition
VAR
	{attribute 'OPC.UA.DA' := '0'}
	_ClassName : STRING := __POUNAME();
END_VAR

{attribute 'monitoring' := 'call'}
PROPERTY ClassName : STRING
GET
ClassName := _ClassName;
END_GET
END_PROPERTY

END_FUNCTION_BLOCK

// ---- StateMachine/UnifiedProgram/Transitions/SuspendedToRunningUnifiedProgramTransition.TcPOU
FUNCTION_BLOCK SuspendedToRunningUnifiedProgramTransition EXTENDS SuspendedToRunningProgramTransition
VAR
	{attribute 'OPC.UA.DA' := '0'}
	_ClassName : STRING := __POUNAME();
END_VAR

{attribute 'monitoring' := 'call'}
PROPERTY ClassName : STRING
GET
ClassName := _ClassName;
END_GET
END_PROPERTY

END_FUNCTION_BLOCK

